(* IEC 61131-3 sources: plc_simulator/services/codesys/POUs, 112 files *)

(* ---- DEP_CalcIdleSlots.st ---- *)
(* ===========================================================================================
 *  DEP_CalcIdleSlots — Idle slot calculation per transporter
 *
 *  Company : Galvatek part of the John Cockerill Group
 *  Author  : Jarmo Piipponen
 *  Created : 25.03.2026
 *
 * -------------------------------------------------------------------------------------------
 *  Reads task queue via VAR_IN_OUT (sandbox or live).
 *  Writes idle slot sets to io_idle_slot per transporter.
 *
 *  ------------------------------------------------------------------------------------------
 *
 *  Changes:
 *
 *
 *
 *)

FUNCTION DEP_CalcIdleSlots : BOOL

(* Introduction of Variables ----------------------------------------------------------------*)

VAR_INPUT
  i_trans                   : INT;
  i_time_s                  : LINT;
END_VAR

VAR_IN_OUT  (* array sizes must match GVL_JC_Constants: 3=MAX_TRANSPORTERS *)
  io_task                   : ARRAY[1..3] OF UDT_JC_TskQueueType;
  io_idle_slot              : ARRAY[1..3] OF UDT_JC_DepIdleSlotSetType;
END_VAR

VAR_EXTERNAL CONSTANT
    MAX_TRANSPORTERS        : INT;
    MAX_UNITS               : INT;
    DEP_MAX_IDLE_SLOTS      : INT;
END_VAR

VAR_EXTERNAL
  g_transporter             : ARRAY[1..MAX_TRANSPORTERS] OF UDT_TransporterStatusType;
END_VAR

VAR
  qi                        : INT;
  si                        : INT;
  cnt                       : INT;
  prev_end                  : LINT;
  prev_sink                 : INT;
  gap_start                 : LINT;
  gap_end                   : LINT;
  HORIZON                   : LINT := 9999999999;
END_VAR

DEP_CalcIdleSlots := FALSE;
IF i_trans < 1 OR i_trans > MAX_TRANSPORTERS THEN RETURN; END_IF;

io_idle_slot[i_trans].Count := 0;
si := 0;
cnt := io_task[i_trans].Count;

prev_end  := i_time_s;
prev_sink := g_transporter[i_trans].CurrentStation;

FOR qi := 1 TO MAX_UNITS DO
  IF qi > cnt THEN EXIT; END_IF;

  gap_start := prev_end;
  gap_end   := io_task[i_trans].Queue[qi].StartTime;

  IF gap_end > gap_start + LINT#1 THEN
    si := si + 1;
    IF si <= DEP_MAX_IDLE_SLOTS THEN
      io_idle_slot[i_trans].Slots[si].StartTime   := gap_start;
      io_idle_slot[i_trans].Slots[si].EndTime     := gap_end;
      io_idle_slot[i_trans].Slots[si].LiftStationTarget := prev_sink;
      io_idle_slot[i_trans].Slots[si].SinkStationTarget := io_task[i_trans].Queue[qi].LiftStationTarget;
    END_IF;
  END_IF;

  prev_end  := io_task[i_trans].Queue[qi].FinishTime;
  prev_sink := io_task[i_trans].Queue[qi].SinkStationTarget;
END_FOR;

si := si + 1;
IF si <= DEP_MAX_IDLE_SLOTS THEN
  io_idle_slot[i_trans].Slots[si].StartTime   := prev_end;
  io_idle_slot[i_trans].Slots[si].EndTime     := HORIZON;
  io_idle_slot[i_trans].Slots[si].LiftStationTarget := prev_sink;
  io_idle_slot[i_trans].Slots[si].SinkStationTarget := 0;
END_IF;

io_idle_slot[i_trans].Count := si;
DEP_CalcIdleSlots := TRUE;

END_FUNCTION

(* ---- DEP_CalcOverlap.st ---- *)
(* ===========================================================================================
 *  DEP_CalcOverlap — Overlap station detection
 *
 *  Company : Galvatek part of the John Cockerill Group
 *  Author  : Jarmo Piipponen
 *  Created : 25.03.2026
 *
 * -------------------------------------------------------------------------------------------
 *  Identifies stations covered by 2+ transporters.
 *  Reads Transporters (read-only config). Writes io_overlap.
 *
 *  ------------------------------------------------------------------------------------------
 *
 *  Changes:
 *
 *
 *
 *)

FUNCTION DEP_CalcOverlap : BOOL

(* Introduction of Variables ----------------------------------------------------------------*)

VAR_IN_OUT
  io_overlap                : UDT_JC_DepOverlapType;
END_VAR

VAR_EXTERNAL CONSTANT
    MAX_TRANSPORTERS        : INT;
    MIN_STATION_INDEX        : INT;
    MAX_STATION_INDEX        : INT;
END_VAR

VAR_EXTERNAL
  Transporters                     : ARRAY[0..MAX_TRANSPORTERS] OF UDT_TransporterType;
END_VAR

VAR
  station_idx               : INT;
  ti                        : INT;
  ai                        : INT;
  cover_count               : INT;
  covered                   : BOOL;
  area                      : UDT_TaskArea;
END_VAR

io_overlap.Count := 0;

FOR station_idx := 0 TO 200 DO
  io_overlap.Flags[station_idx] := FALSE;
END_FOR;

FOR station_idx := MIN_STATION_INDEX TO MAX_STATION_INDEX DO
  cover_count := 0;

  FOR ti := 1 TO MAX_TRANSPORTERS DO
    covered := FALSE;
    FOR ai := 1 TO 4 DO
      IF NOT covered THEN
        area := Transporters[ti].TaskArea[ai];
        IF (area.MinLift > 0 AND station_idx >= area.MinLift AND station_idx <= area.MaxLift)
           OR (area.MinSink > 0 AND station_idx >= area.MinSink AND station_idx <= area.MaxSink) THEN
          covered := TRUE;
        END_IF;
      END_IF;
    END_FOR;
    IF covered THEN
      cover_count := cover_count + 1;
    END_IF;
  END_FOR;

  IF cover_count >= 2 THEN
    io_overlap.Flags[station_idx] := TRUE;
    io_overlap.Count := io_overlap.Count + 1;
  END_IF;
END_FOR;

DEP_CalcOverlap := TRUE;

END_FUNCTION

(* ---- DEP_FC_CalcIdleSlots.st ---- *)
(* ===========================================================================================
 *  DEP_FC_CalcIdleSlots — Idle slot calculation per transporter
 *
 *  Company : Galvatek part of the John Cockerill Group
 *  Author  : Jarmo Piipponen
 *  Created : 25.03.2026
 *
 * -------------------------------------------------------------------------------------------
 *  Reads task queue via VAR_IN_OUT (sandbox or live).
 *  Writes idle slot sets to ioIdleSlot per transporter.
 *
 *  ------------------------------------------------------------------------------------------
 *
 *  Changes:
 *
 *
 *
 *)

FUNCTION DEP_FC_CalcIdleSlots : BOOL

(* Introduction of Variables ----------------------------------------------------------------*)

VAR_INPUT
  iTrans                   : INT;
  iTimeS                  : LINT;
END_VAR

VAR_IN_OUT  (* array sizes must match GVL_JC_Constants: 3=MAX_TRANSPORTERS *)
  ioTask                   : ARRAY[1..3] OF UDT_JC_TskQueueType;
  ioIdleSlot              : ARRAY[1..3] OF UDT_JC_DepIdleSlotSetType;
END_VAR

VAR_EXTERNAL CONSTANT
    MAX_TRANSPORTERS        : INT;
    MAX_UNITS               : INT;
    DEP_MAX_IDLE_SLOTS      : INT;
END_VAR

VAR_EXTERNAL
  TransporterStatus             : ARRAY[1..MAX_TRANSPORTERS] OF UDT_TransporterStatusType;
END_VAR

VAR
  vQi                        : INT;
  vSi                        : INT;
  vCnt                       : INT;
  vPrevEnd                  : LINT;
  vPrevSink                 : INT;
  vGapStart                 : LINT;
  vGapEnd                   : LINT;
  vHorizon                   : LINT := 9999999999;
END_VAR

DEP_FC_CalcIdleSlots := FALSE;
IF iTrans < 1 OR iTrans > MAX_TRANSPORTERS THEN RETURN; END_IF;

ioIdleSlot[iTrans].Count := 0;
vSi := 0;
vCnt := ioTask[iTrans].Count;

vPrevEnd  := iTimeS;
vPrevSink := TransporterStatus[iTrans].CurrentStation;

FOR vQi := 1 TO MAX_UNITS DO
  IF vQi > vCnt THEN EXIT; END_IF;

  vGapStart := vPrevEnd;
  vGapEnd   := ioTask[iTrans].Queue[vQi].StartTime;

  IF vGapEnd > vGapStart + LINT#1 THEN
    vSi := vSi + 1;
    IF vSi <= DEP_MAX_IDLE_SLOTS THEN
      ioIdleSlot[iTrans].Slots[vSi].StartTime   := vGapStart;
      ioIdleSlot[iTrans].Slots[vSi].EndTime     := vGapEnd;
      ioIdleSlot[iTrans].Slots[vSi].LiftStationTarget := vPrevSink;
      ioIdleSlot[iTrans].Slots[vSi].SinkStationTarget := ioTask[iTrans].Queue[vQi].LiftStationTarget;
    END_IF;
  END_IF;

  vPrevEnd  := ioTask[iTrans].Queue[vQi].FinishTime;
  vPrevSink := ioTask[iTrans].Queue[vQi].SinkStationTarget;
END_FOR;

vSi := vSi + 1;
IF vSi <= DEP_MAX_IDLE_SLOTS THEN
  ioIdleSlot[iTrans].Slots[vSi].StartTime   := vPrevEnd;
  ioIdleSlot[iTrans].Slots[vSi].EndTime     := vHorizon;
  ioIdleSlot[iTrans].Slots[vSi].LiftStationTarget := vPrevSink;
  ioIdleSlot[iTrans].Slots[vSi].SinkStationTarget := 0;
END_IF;

ioIdleSlot[iTrans].Count := vSi;
DEP_FC_CalcIdleSlots := TRUE;

END_FUNCTION

(* ---- DEP_FC_CalcOverlap.st ---- *)
(* ===========================================================================================
 *  DEP_FC_CalcOverlap — Overlap station detection
 *
 *  Company : Galvatek part of the John Cockerill Group
 *  Author  : Jarmo Piipponen
 *  Created : 25.03.2026
 *
 * -------------------------------------------------------------------------------------------
 *  Identifies stations vCovered by 2+ transporters.
 *  Reads Transporters (read-only config). Writes ioOverlap.
 *
 *  ------------------------------------------------------------------------------------------
 *
 *  Changes:
 *
 *
 *
 *)

FUNCTION DEP_FC_CalcOverlap : BOOL

(* Introduction of Variables ----------------------------------------------------------------*)

VAR_IN_OUT
  ioOverlap                : UDT_JC_DepOverlapType;
END_VAR

VAR_EXTERNAL CONSTANT
    MAX_TRANSPORTERS        : INT;
    MIN_STATION_INDEX        : INT;
    MAX_STATION_INDEX        : INT;
END_VAR

VAR_EXTERNAL
  Transporters                     : ARRAY[0..MAX_TRANSPORTERS] OF UDT_TransporterType;
END_VAR

VAR
  vStationIdx               : INT;
  vTi                        : INT;
  vAi                        : INT;
  vCoverCount               : INT;
  vCovered                   : BOOL;
  vArea                      : UDT_TaskAreaType;
END_VAR

ioOverlap.Count := 0;

FOR vStationIdx := 0 TO 200 DO
  ioOverlap.Flags[vStationIdx] := FALSE;
END_FOR;

FOR vStationIdx := MIN_STATION_INDEX TO MAX_STATION_INDEX DO
  vCoverCount := 0;

  FOR vTi := 1 TO MAX_TRANSPORTERS DO
    vCovered := FALSE;
    FOR vAi := 1 TO 4 DO
      IF NOT vCovered THEN
        vArea := Transporters[vTi].TaskArea[vAi];
        IF (vArea.MinLift > 0 AND vStationIdx >= vArea.MinLift AND vStationIdx <= vArea.MaxLift)
           OR (vArea.MinSink > 0 AND vStationIdx >= vArea.MinSink AND vStationIdx <= vArea.MaxSink) THEN
          vCovered := TRUE;
        END_IF;
      END_IF;
    END_FOR;
    IF vCovered THEN
      vCoverCount := vCoverCount + 1;
    END_IF;
  END_FOR;

  IF vCoverCount >= 2 THEN
    ioOverlap.Flags[vStationIdx] := TRUE;
    ioOverlap.Count := ioOverlap.Count + 1;
  END_IF;
END_FOR;

DEP_FC_CalcOverlap := TRUE;

END_FUNCTION

(* ---- DEP_FC_FitTaskToSlot.st ---- *)
(* ===========================================================================================
 *  DEP_FC_FitTaskToSlot — Fit a departure task into idle slots
 *
 *  Company : Galvatek part of the John Cockerill Group
 *  Author  : Jarmo Piipponen
 *  Created : 25.03.2026
 *
 * -------------------------------------------------------------------------------------------
 *  Reads idle slots and move times.
 *  Returns fit result via VAR_OUTPUT.
 *
 *  ------------------------------------------------------------------------------------------
 *
 *  Changes:
 *
 *
 *
 *)

FUNCTION DEP_FC_FitTaskToSlot : BOOL

(* Introduction of Variables ----------------------------------------------------------------*)

VAR_INPUT
  iLiftStn                : INT;
  iSinkStn                : INT;
  iTransId                : INT;
  iTaskStart              : LINT;
  iTaskEnd                : LINT;
  iShiftS                 : REAL;
  iCalcTimeS             : DINT;
  iMinTimeS              : DINT;
  iMaxTimeS              : DINT;
  iFlexFactor             : REAL;
  iMarginS                : REAL;
  iConflictMarginS       : REAL;
END_VAR

VAR_IN_OUT  (* array sizes must match GVL_JC_Constants: 3=MAX_TRANSPORTERS *)
  ioIdleSlot              : ARRAY[1..3] OF UDT_JC_DepIdleSlotSetType;
  ioOResult                  : UDT_JC_DepFitResultType;
END_VAR

VAR_EXTERNAL CONSTANT
    MAX_TRANSPORTERS        : INT;
    DEP_MAX_IDLE_SLOTS      : INT;
    SCH_DISPATCH_MARGIN_S   : REAL;
END_VAR

VAR_EXTERNAL
  Move                    : ARRAY[1..MAX_TRANSPORTERS] OF UDT_JC_MoveTimesType;
END_VAR

VAR
  vSi                        : INT;
  vSlotCnt                  : INT;
  vSlotStart                : LINT;
  vSlotEnd                  : LINT;
  vFromStn                  : INT;
  vToStn                    : INT;
  vTravelTo                 : REAL;
  vTravelFrom               : REAL;
  vEarliest                  : LINT;
  vLatest                    : LINT;
  vTaskDur                  : LINT;
  vDelay                     : REAL;
  vFlexUp                   : REAL;
  vCappedFlex               : REAL;
  vBestDelay                : REAL;
  vBestSlot                 : INT;
  vFound                     : BOOL;
  vOverflowBestDelay       : REAL;
  vOverflowBestSlot        : INT;
  vTmpMove                  : UDT_JC_MoveTimesType;
  vTotalDelay               : REAL;
END_VAR

ioOResult.Fits         := FALSE;
ioOResult.DelayTime    := 0;
ioOResult.NeedExtraTime := 0;
ioOResult.TaskEndTime  := 0;
ioOResult.SlotIdx      := 0;
ioOResult.OverflowSlotIdx := 0;
ioOResult.TransporterId := iTransId;
DEP_FC_FitTaskToSlot := FALSE;

IF iTransId < 1 OR iTransId > MAX_TRANSPORTERS THEN RETURN; END_IF;

vTaskDur   := iTaskEnd - iTaskStart;
(* Absolute cap: flex based on full (max - min) range, not (max - calc).
   This prevents cumulative drift when CalcTime is adjusted across rounds. *)
vFlexUp    := DINT_TO_REAL(iMaxTimeS - iMinTimeS);
  IF vFlexUp < 0.0 THEN vFlexUp := 0.0; END_IF;
vCappedFlex := vFlexUp * iFlexFactor;

vSlotCnt   := ioIdleSlot[iTransId].Count;
vBestDelay := 1.0E9;
vBestSlot  := 0;
vFound      := FALSE;
vOverflowBestDelay := 1.0E9;
vOverflowBestSlot  := 0;

vTmpMove := Move[iTransId];
FOR vSi := 1 TO DEP_MAX_IDLE_SLOTS DO
  IF vSi > vSlotCnt THEN EXIT; END_IF;

  vSlotStart := ioIdleSlot[iTransId].Slots[vSi].StartTime;
  vSlotEnd   := ioIdleSlot[iTransId].Slots[vSi].EndTime;

  vFromStn := ioIdleSlot[iTransId].Slots[vSi].LiftStationTarget;
  vTravelTo := 0.0;
  IF vFromStn > 0 AND vFromStn <> iLiftStn THEN
    vTravelTo := STC_FC_CalcHorizontalTravel(iFromStn := vFromStn, iToStn := iLiftStn, iMove := vTmpMove);
  END_IF;

  vToStn := ioIdleSlot[iTransId].Slots[vSi].SinkStationTarget;
  vTravelFrom := 0.0;
  IF vToStn > 0 AND vToStn <> iSinkStn THEN
    vTravelFrom := STC_FC_CalcHorizontalTravel(iFromStn := iSinkStn, iToStn := vToStn, iMove := vTmpMove);
  END_IF;

  (* vEarliest = max(transporter arrival, task readiness) + conflict margin *)
  IF (vSlotStart + REAL_TO_LINT(vTravelTo)) > (iTaskStart + REAL_TO_LINT(iShiftS)) THEN
    vEarliest := vSlotStart + REAL_TO_LINT(vTravelTo + iConflictMarginS);
  ELSE
    vEarliest := iTaskStart + REAL_TO_LINT(iShiftS + iConflictMarginS);
  END_IF;

  IF vSlotEnd > LINT#9000000000 THEN
    vLatest := LINT#9000000000;
  ELSE
    vLatest := vSlotEnd - REAL_TO_LINT(vTravelFrom + SCH_DISPATCH_MARGIN_S);
  END_IF;

  IF vEarliest + vTaskDur <= vLatest THEN
    vDelay := LINT_TO_REAL(vEarliest - iTaskStart) - iShiftS;
  IF vDelay < 0.0 THEN vDelay := 0.0; END_IF;
    vTotalDelay := iShiftS + vDelay;

    IF vTotalDelay <= iMarginS OR vTotalDelay <= vCappedFlex + 1.0 THEN
      IF vDelay < vBestDelay THEN
        vBestDelay := vDelay;
        vBestSlot  := vSi;
        vFound      := TRUE;
      END_IF;
    ELSE
      IF vDelay < vOverflowBestDelay THEN
        vOverflowBestDelay := vDelay;
        vOverflowBestSlot  := vSi;
      END_IF;
    END_IF;
  END_IF;
END_FOR;

IF vFound THEN
  ioOResult.Fits      := TRUE;
  ioOResult.DelayTime := REAL_TO_DINT(vBestDelay);
  ioOResult.SlotIdx   := vBestSlot;
  ioOResult.TaskEndTime := iTaskStart + REAL_TO_LINT(iShiftS + vBestDelay) + vTaskDur;
  ioOResult.NeedExtraTime := 0;
ELSE
  ioOResult.Fits := FALSE;
  IF vOverflowBestDelay < 1.0E8 THEN
    ioOResult.DelayTime     := REAL_TO_DINT(vOverflowBestDelay);
    ioOResult.NeedExtraTime := REAL_TO_DINT(iShiftS + vOverflowBestDelay - vCappedFlex);
  IF ioOResult.NeedExtraTime < 0 THEN ioOResult.NeedExtraTime := 0; END_IF;
    ioOResult.OverflowSlotIdx := vOverflowBestSlot;
  ELSE
    ioOResult.NeedExtraTime := 0;
  END_IF;
END_IF;

DEP_FC_FitTaskToSlot := TRUE;

END_FUNCTION

(* ---- DEP_FC_OverlapDelay.st ---- *)
(* ===========================================================================================
 *  DEP_FC_OverlapDelay — Overlap conflict vDelay calculation
 *
 *  Company : Galvatek part of the John Cockerill Group
 *  Author  : Jarmo Piipponen
 *  Created : 25.03.2026
 *
 * -------------------------------------------------------------------------------------------
 *  Returns vDelay vNeeded to avoid overlap conflicts.
 *  Reads task queues via ioTask (sandbox or live).
 *
 *  ------------------------------------------------------------------------------------------
 *
 *  Changes:
 *
 *
 *
 *)

FUNCTION DEP_FC_OverlapDelay : REAL   (* returns delay_s, 0 = no conflict *)

(* Introduction of Variables ----------------------------------------------------------------*)

VAR_INPUT
  iLiftStn                : INT;
  iSinkStn                : INT;
  iTransId                : INT;
  iTaskStart              : LINT;
  iTaskEnd                : LINT;
  iMarginS                : REAL;
END_VAR

VAR_IN_OUT  (* array sizes must match GVL_JC_Constants: 3=MAX_TRANSPORTERS *)
  ioTask                   : ARRAY[1..3] OF UDT_JC_TskQueueType;
  ioOverlap                : UDT_JC_DepOverlapType;
END_VAR

VAR_EXTERNAL CONSTANT
    MAX_TRANSPORTERS        : INT;
    MAX_UNITS               : INT;
    DEP_MAX_DELAY_ACTS      : INT;
END_VAR

VAR
  vLiftIsOverlap           : BOOL;
  vSinkIsOverlap           : BOOL;
  vRound                     : INT;
  vTi                        : INT;
  vQi                        : INT;
  vMaxConf                  : REAL;
  vTStart                   : LINT;
  vTEnd                     : LINT;
  vEStart                   : LINT;
  vEEnd                     : LINT;
  vELift                    : INT;
  vESink                    : INT;
  vHasOvlp                  : BOOL;
  vNeeded                    : REAL;
  vDelay                     : REAL;
END_VAR

vDelay := 0.0;

IF iLiftStn >= 0 AND iLiftStn <= 200 THEN
  vLiftIsOverlap := ioOverlap.Flags[iLiftStn];
ELSE
  vLiftIsOverlap := FALSE;
END_IF;
IF iSinkStn >= 0 AND iSinkStn <= 200 THEN
  vSinkIsOverlap := ioOverlap.Flags[iSinkStn];
ELSE
  vSinkIsOverlap := FALSE;
END_IF;

IF NOT vLiftIsOverlap AND NOT vSinkIsOverlap THEN
  DEP_FC_OverlapDelay := 0.0;
  RETURN;
END_IF;

FOR vRound := 1 TO DEP_MAX_DELAY_ACTS DO
  vMaxConf := 0.0;
  vTStart  := iTaskStart + REAL_TO_LINT(vDelay);
  vTEnd    := iTaskEnd + REAL_TO_LINT(vDelay);

  FOR vTi := 1 TO MAX_TRANSPORTERS DO
    IF vTi <> iTransId THEN
      FOR vQi := 1 TO MAX_UNITS DO
        IF vQi > ioTask[vTi].Count THEN EXIT; END_IF;

        vELift  := ioTask[vTi].Queue[vQi].LiftStationTarget;
        vESink  := ioTask[vTi].Queue[vQi].SinkStationTarget;
        vEStart := ioTask[vTi].Queue[vQi].StartTime;
        vEEnd   := ioTask[vTi].Queue[vQi].FinishTime;

        vHasOvlp := FALSE;
        IF vELift >= 0 AND vELift <= 200 THEN
  IF ioOverlap.Flags[vELift] THEN vHasOvlp := TRUE; END_IF;
        END_IF;
        IF NOT vHasOvlp AND vESink >= 0 AND vESink <= 200 THEN
  IF ioOverlap.Flags[vESink] THEN vHasOvlp := TRUE; END_IF;
        END_IF;

        IF vHasOvlp THEN
          IF vTStart < (vEEnd + REAL_TO_LINT(iMarginS)) AND vTEnd > (vEStart - REAL_TO_LINT(iMarginS)) THEN
            vNeeded := LINT_TO_REAL(vEEnd - vTStart) + iMarginS;
  IF vNeeded > vMaxConf THEN vMaxConf := vNeeded; END_IF;
          END_IF;
        END_IF;

      END_FOR;
    END_IF;
  END_FOR;

  IF vMaxConf <= 0.0 THEN EXIT; END_IF;
  vDelay := vDelay + vMaxConf;
END_FOR;

DEP_FC_OverlapDelay := vDelay;

END_FUNCTION

(* ---- DEP_FC_Sandbox.st ---- *)
(* ===========================================================================================
 *  DEP_FC_Sandbox — Sandbox snapshot / restore / clear
 *
 *  Company : Galvatek part of the John Cockerill Group
 *  Author  : Jarmo Piipponen
 *  Created : 25.03.2026
 *
 * -------------------------------------------------------------------------------------------
 *  Copies batch and program data between live globals and
 *  DEP workspace arrays via VAR_IN_OUT.
 *  Schedule is NOT copied — DEP calculates it fresh (phases 1000+i).
 *  Task queues are NOT copied — DEP rebuilds them (phases 2000+).
 *
 *  Commands:
 *  1 = SNAPSHOT  — live batch+program → workspace
 *  2 = RESTORE   — workspace batch+program → live
 *  3 = CLEAR     — noop for array-based workspace
 *
 *  ------------------------------------------------------------------------------------------
 *
 *  Changes:
 *
 *
 *
 *)

FUNCTION DEP_FC_Sandbox : BOOL

(* Introduction of Variables ----------------------------------------------------------------*)

VAR_INPUT
  iCmd                     : INT;
END_VAR

VAR_IN_OUT  (* array sizes must match GVL_JC_Constants: 10=MAX_UNITS, 3=MAX_TRANSPORTERS *)
  ioWkSchedule            : ARRAY[1..10] OF UDT_JC_TskScheduleType;
  ioWkBatch               : ARRAY[1..10] OF UDT_BatchType;
  ioWkProgram             : ARRAY[1..10] OF UDT_TreatmentProgramType;
  ioWkTask                : ARRAY[1..3] OF UDT_JC_TskQueueType;
END_VAR

VAR_EXTERNAL CONSTANT
    MAX_TRANSPORTERS        : INT;
    MAX_UNITS               : INT;
END_VAR

VAR_EXTERNAL
  Schedule                : ARRAY[1..MAX_UNITS] OF UDT_JC_TskScheduleType;
  Batch                   : ARRAY[1..MAX_UNITS] OF UDT_BatchType;
  TreatmentPrograms                 : ARRAY[1..MAX_UNITS] OF UDT_TreatmentProgramType;
  Task                    : ARRAY[1..MAX_TRANSPORTERS] OF UDT_JC_TskQueueType;
END_VAR

VAR
  vUi                        : INT;
END_VAR

DEP_FC_Sandbox := TRUE;

IF iCmd = 1 THEN
  (* SNAPSHOT: clear workspace, then copy live batch+program *)
  FOR vUi := 1 TO MAX_UNITS DO
    ioWkSchedule[vUi].StageCount := 0;
    ioWkBatch[vUi]    := Batch[vUi];
    ioWkProgram[vUi]  := TreatmentPrograms[vUi];
  END_FOR;
  FOR vUi := 1 TO MAX_TRANSPORTERS DO
    ioWkTask[vUi].Count := 0;
  END_FOR;
ELSIF iCmd = 2 THEN
  (* RESTORE: workspace batch+program → live (for REJECT rollback) *)
  FOR vUi := 1 TO MAX_UNITS DO
    IF ioWkBatch[vUi].BatchCode > 0 THEN
      Batch[vUi] := ioWkBatch[vUi];
    END_IF;
    IF ioWkProgram[vUi].ProgramId > 0 THEN
      TreatmentPrograms[vUi] := ioWkProgram[vUi];
    END_IF;
  END_FOR;
ELSIF iCmd = 3 THEN
  ;  (* CLEAR: nothing needed *)

END_IF;

END_FUNCTION

(* ---- DEP_FitTaskToSlot.st ---- *)
(* ===========================================================================================
 *  DEP_FitTaskToSlot — Fit a departure task into idle slots
 *
 *  Company : Galvatek part of the John Cockerill Group
 *  Author  : Jarmo Piipponen
 *  Created : 25.03.2026
 *
 * -------------------------------------------------------------------------------------------
 *  Reads idle slots and move times.
 *  Returns fit result via VAR_OUTPUT.
 *
 *  ------------------------------------------------------------------------------------------
 *
 *  Changes:
 *
 *
 *
 *)

FUNCTION DEP_FitTaskToSlot : BOOL

(* Introduction of Variables ----------------------------------------------------------------*)

VAR_INPUT
  i_lift_stn                : INT;
  i_sink_stn                : INT;
  i_trans_id                : INT;
  i_task_start              : LINT;
  i_task_end                : LINT;
  i_shift_s                 : REAL;
  i_calc_time_s             : DINT;
  i_min_time_s              : DINT;
  i_max_time_s              : DINT;
  i_flex_factor             : REAL;
  i_margin_s                : REAL;
  i_conflict_margin_s       : REAL;
END_VAR

VAR_IN_OUT  (* array sizes must match GVL_JC_Constants: 3=MAX_TRANSPORTERS *)
  io_idle_slot              : ARRAY[1..3] OF UDT_JC_DepIdleSlotSetType;
  o_result                  : UDT_JC_DepFitResultType;
END_VAR

VAR_EXTERNAL CONSTANT
    MAX_TRANSPORTERS        : INT;
    DEP_MAX_IDLE_SLOTS      : INT;
    SCH_DISPATCH_MARGIN_S   : REAL;
END_VAR

VAR_EXTERNAL
  g_move                    : ARRAY[1..MAX_TRANSPORTERS] OF UDT_JC_MoveTimesType;
END_VAR

VAR
  si                        : INT;
  slot_cnt                  : INT;
  slot_start                : LINT;
  slot_end                  : LINT;
  from_stn                  : INT;
  to_stn                    : INT;
  travel_to                 : REAL;
  travel_from               : REAL;
  earliest                  : LINT;
  latest                    : LINT;
  task_dur                  : LINT;
  delay                     : REAL;
  flex_up                   : REAL;
  capped_flex               : REAL;
  best_delay                : REAL;
  best_slot                 : INT;
  found                     : BOOL;
  overflow_best_delay       : REAL;
  overflow_best_slot        : INT;
  tmp_move                  : UDT_JC_MoveTimesType;
  total_delay               : REAL;
END_VAR

o_result.Fits         := FALSE;
o_result.DelayTime    := 0;
o_result.NeedExtraTime := 0;
o_result.TaskEndTime  := 0;
o_result.SlotIdx      := 0;
o_result.OverflowSlotIdx := 0;
o_result.TransporterId := i_trans_id;
DEP_FitTaskToSlot := FALSE;

IF i_trans_id < 1 OR i_trans_id > MAX_TRANSPORTERS THEN RETURN; END_IF;

task_dur   := i_task_end - i_task_start;
(* Absolute cap: flex based on full (max - min) range, not (max - calc).
   This prevents cumulative drift when CalcTime is adjusted across rounds. *)
flex_up    := DINT_TO_REAL(i_max_time_s - i_min_time_s);
  IF flex_up < 0.0 THEN flex_up := 0.0; END_IF;
capped_flex := flex_up * i_flex_factor;

slot_cnt   := io_idle_slot[i_trans_id].Count;
best_delay := 1.0E9;
best_slot  := 0;
found      := FALSE;
overflow_best_delay := 1.0E9;
overflow_best_slot  := 0;

tmp_move := g_move[i_trans_id];
FOR si := 1 TO DEP_MAX_IDLE_SLOTS DO
  IF si > slot_cnt THEN EXIT; END_IF;

  slot_start := io_idle_slot[i_trans_id].Slots[si].StartTime;
  slot_end   := io_idle_slot[i_trans_id].Slots[si].EndTime;

  from_stn := io_idle_slot[i_trans_id].Slots[si].LiftStationTarget;
  travel_to := 0.0;
  IF from_stn > 0 AND from_stn <> i_lift_stn THEN
    travel_to := STC_CalcHorizontalTravel(i_from_stn := from_stn, i_to_stn := i_lift_stn, i_move := tmp_move);
  END_IF;

  to_stn := io_idle_slot[i_trans_id].Slots[si].SinkStationTarget;
  travel_from := 0.0;
  IF to_stn > 0 AND to_stn <> i_sink_stn THEN
    travel_from := STC_CalcHorizontalTravel(i_from_stn := i_sink_stn, i_to_stn := to_stn, i_move := tmp_move);
  END_IF;

  (* earliest = max(transporter arrival, task readiness) + conflict margin *)
  IF (slot_start + REAL_TO_LINT(travel_to)) > (i_task_start + REAL_TO_LINT(i_shift_s)) THEN
    earliest := slot_start + REAL_TO_LINT(travel_to + i_conflict_margin_s);
  ELSE
    earliest := i_task_start + REAL_TO_LINT(i_shift_s + i_conflict_margin_s);
  END_IF;

  IF slot_end > LINT#9000000000 THEN
    latest := LINT#9000000000;
  ELSE
    latest := slot_end - REAL_TO_LINT(travel_from + SCH_DISPATCH_MARGIN_S);
  END_IF;

  IF earliest + task_dur <= latest THEN
    delay := LINT_TO_REAL(earliest - i_task_start) - i_shift_s;
  IF delay < 0.0 THEN delay := 0.0; END_IF;
    total_delay := i_shift_s + delay;

    IF total_delay <= i_margin_s OR total_delay <= capped_flex + 1.0 THEN
      IF delay < best_delay THEN
        best_delay := delay;
        best_slot  := si;
        found      := TRUE;
      END_IF;
    ELSE
      IF delay < overflow_best_delay THEN
        overflow_best_delay := delay;
        overflow_best_slot  := si;
      END_IF;
    END_IF;
  END_IF;
END_FOR;

IF found THEN
  o_result.Fits      := TRUE;
  o_result.DelayTime := REAL_TO_DINT(best_delay);
  o_result.SlotIdx   := best_slot;
  o_result.TaskEndTime := i_task_start + REAL_TO_LINT(i_shift_s + best_delay) + task_dur;
  o_result.NeedExtraTime := 0;
ELSE
  o_result.Fits := FALSE;
  IF overflow_best_delay < 1.0E8 THEN
    o_result.DelayTime     := REAL_TO_DINT(overflow_best_delay);
    o_result.NeedExtraTime := REAL_TO_DINT(i_shift_s + overflow_best_delay - capped_flex);
  IF o_result.NeedExtraTime < 0 THEN o_result.NeedExtraTime := 0; END_IF;
    o_result.OverflowSlotIdx := overflow_best_slot;
  ELSE
    o_result.NeedExtraTime := 0;
  END_IF;
END_IF;

DEP_FitTaskToSlot := TRUE;

END_FUNCTION

(* ---- DEP_OverlapDelay.st ---- *)
(* ===========================================================================================
 *  DEP_OverlapDelay — Overlap conflict delay calculation
 *
 *  Company : Galvatek part of the John Cockerill Group
 *  Author  : Jarmo Piipponen
 *  Created : 25.03.2026
 *
 * -------------------------------------------------------------------------------------------
 *  Returns delay needed to avoid overlap conflicts.
 *  Reads task queues via io_task (sandbox or live).
 *
 *  ------------------------------------------------------------------------------------------
 *
 *  Changes:
 *
 *
 *
 *)

FUNCTION DEP_OverlapDelay : REAL   (* returns delay_s, 0 = no conflict *)

(* Introduction of Variables ----------------------------------------------------------------*)

VAR_INPUT
  i_lift_stn                : INT;
  i_sink_stn                : INT;
  i_trans_id                : INT;
  i_task_start              : LINT;
  i_task_end                : LINT;
  i_margin_s                : REAL;
END_VAR

VAR_IN_OUT  (* array sizes must match GVL_JC_Constants: 3=MAX_TRANSPORTERS *)
  io_task                   : ARRAY[1..3] OF UDT_JC_TskQueueType;
  io_overlap                : UDT_JC_DepOverlapType;
END_VAR

VAR_EXTERNAL CONSTANT
    MAX_TRANSPORTERS        : INT;
    MAX_UNITS               : INT;
    DEP_MAX_DELAY_ACTS      : INT;
END_VAR

VAR
  lift_is_overlap           : BOOL;
  sink_is_overlap           : BOOL;
  round                     : INT;
  ti                        : INT;
  qi                        : INT;
  max_conf                  : REAL;
  t_start                   : LINT;
  t_end                     : LINT;
  e_start                   : LINT;
  e_end                     : LINT;
  e_lift                    : INT;
  e_sink                    : INT;
  has_ovlp                  : BOOL;
  needed                    : REAL;
  delay                     : REAL;
END_VAR

delay := 0.0;

IF i_lift_stn >= 0 AND i_lift_stn <= 200 THEN
  lift_is_overlap := io_overlap.Flags[i_lift_stn];
ELSE
  lift_is_overlap := FALSE;
END_IF;
IF i_sink_stn >= 0 AND i_sink_stn <= 200 THEN
  sink_is_overlap := io_overlap.Flags[i_sink_stn];
ELSE
  sink_is_overlap := FALSE;
END_IF;

IF NOT lift_is_overlap AND NOT sink_is_overlap THEN
  DEP_OverlapDelay := 0.0;
  RETURN;
END_IF;

FOR round := 1 TO DEP_MAX_DELAY_ACTS DO
  max_conf := 0.0;
  t_start  := i_task_start + REAL_TO_LINT(delay);
  t_end    := i_task_end + REAL_TO_LINT(delay);

  FOR ti := 1 TO MAX_TRANSPORTERS DO
    IF ti <> i_trans_id THEN
      FOR qi := 1 TO MAX_UNITS DO
        IF qi > io_task[ti].Count THEN EXIT; END_IF;

        e_lift  := io_task[ti].Queue[qi].LiftStationTarget;
        e_sink  := io_task[ti].Queue[qi].SinkStationTarget;
        e_start := io_task[ti].Queue[qi].StartTime;
        e_end   := io_task[ti].Queue[qi].FinishTime;

        has_ovlp := FALSE;
        IF e_lift >= 0 AND e_lift <= 200 THEN
  IF io_overlap.Flags[e_lift] THEN has_ovlp := TRUE; END_IF;
        END_IF;
        IF NOT has_ovlp AND e_sink >= 0 AND e_sink <= 200 THEN
  IF io_overlap.Flags[e_sink] THEN has_ovlp := TRUE; END_IF;
        END_IF;

        IF has_ovlp THEN
          IF t_start < (e_end + REAL_TO_LINT(i_margin_s)) AND t_end > (e_start - REAL_TO_LINT(i_margin_s)) THEN
            needed := LINT_TO_REAL(e_end - t_start) + i_margin_s;
  IF needed > max_conf THEN max_conf := needed; END_IF;
          END_IF;
        END_IF;

      END_FOR;
    END_IF;
  END_FOR;

  IF max_conf <= 0.0 THEN EXIT; END_IF;
  delay := delay + max_conf;
END_FOR;

DEP_OverlapDelay := delay;

END_FUNCTION

(* ---- DEP_Sandbox.st ---- *)
(* ===========================================================================================
 *  DEP_Sandbox — Sandbox snapshot / restore / clear
 *
 *  Company : Galvatek part of the John Cockerill Group
 *  Author  : Jarmo Piipponen
 *  Created : 25.03.2026
 *
 * -------------------------------------------------------------------------------------------
 *  Copies batch and program data between live globals and
 *  DEP workspace arrays via VAR_IN_OUT.
 *  Schedule is NOT copied — DEP calculates it fresh (phases 1000+i).
 *  Task queues are NOT copied — DEP rebuilds them (phases 2000+).
 *
 *  Commands:
 *  1 = SNAPSHOT  — live batch+program → workspace
 *  2 = RESTORE   — workspace batch+program → live
 *  3 = CLEAR     — noop for array-based workspace
 *
 *  ------------------------------------------------------------------------------------------
 *
 *  Changes:
 *
 *
 *
 *)

FUNCTION DEP_Sandbox : BOOL

(* Introduction of Variables ----------------------------------------------------------------*)

VAR_INPUT
  i_cmd                     : INT;
END_VAR

VAR_IN_OUT  (* array sizes must match GVL_JC_Constants: 10=MAX_UNITS, 3=MAX_TRANSPORTERS *)
  io_wk_schedule            : ARRAY[1..10] OF UDT_JC_TskScheduleType;
  io_wk_batch               : ARRAY[1..10] OF UDT_BatchType;
  io_wk_program             : ARRAY[1..10] OF UDT_TreatmentProgramType;
  io_wk_task                : ARRAY[1..3] OF UDT_JC_TskQueueType;
END_VAR

VAR_EXTERNAL CONSTANT
    MAX_TRANSPORTERS        : INT;
    MAX_UNITS               : INT;
END_VAR

VAR_EXTERNAL
  g_schedule                : ARRAY[1..MAX_UNITS] OF UDT_JC_TskScheduleType;
  g_batch                   : ARRAY[1..MAX_UNITS] OF UDT_BatchType;
  TreatmentPrograms                 : ARRAY[1..MAX_UNITS] OF UDT_TreatmentProgramType;
  g_task                    : ARRAY[1..MAX_TRANSPORTERS] OF UDT_JC_TskQueueType;
END_VAR

VAR
  ui                        : INT;
END_VAR

DEP_Sandbox := TRUE;

IF i_cmd = 1 THEN
  (* SNAPSHOT: clear workspace, then copy live batch+program *)
  FOR ui := 1 TO MAX_UNITS DO
    io_wk_schedule[ui].StageCount := 0;
    io_wk_batch[ui]    := g_batch[ui];
    io_wk_program[ui]  := TreatmentPrograms[ui];
  END_FOR;
  FOR ui := 1 TO MAX_TRANSPORTERS DO
    io_wk_task[ui].Count := 0;
  END_FOR;
ELSIF i_cmd = 2 THEN
  (* RESTORE: workspace batch+program → live (for REJECT rollback) *)
  FOR ui := 1 TO MAX_UNITS DO
    IF io_wk_batch[ui].BatchCode > 0 THEN
      g_batch[ui] := io_wk_batch[ui];
    END_IF;
    IF io_wk_program[ui].ProgramId > 0 THEN
      TreatmentPrograms[ui] := io_wk_program[ui];
    END_IF;
  END_FOR;
ELSIF i_cmd = 3 THEN
  ;  (* CLEAR: nothing needed *)

END_IF;

END_FUNCTION

(* ---- FC_DEP_CalcIdleSlots.st ---- *)
(* ===========================================================================================
 *  FC_DEP_CalcIdleSlots — Idle slot calculation per transporter
 *
 *  Company : Galvatek part of the John Cockerill Group
 *  Author  : Jarmo Piipponen
 *  Created : 25.03.2026
 *
 * -------------------------------------------------------------------------------------------
 *  Reads task queue via VAR_IN_OUT (sandbox or live).
 *  Writes idle slot sets to ioIdleSlot per transporter.
 *
 *  ------------------------------------------------------------------------------------------
 *
 *  Changes:
 *
 *
 *
 *)

FUNCTION FC_DEP_CalcIdleSlots : BOOL

(* Introduction of Variables ----------------------------------------------------------------*)

VAR_INPUT
  iTrans                   : INT;
  iTimeS                  : LINT;
END_VAR

VAR_IN_OUT  (* array sizes must match GVL_JC_Constants: 3=MAX_TRANSPORTERS *)
  ioTask                   : ARRAY[1..3] OF UDT_JC_TskQueueType;
  ioIdleSlot              : ARRAY[1..3] OF UDT_JC_DepIdleSlotSetType;
END_VAR

VAR_EXTERNAL CONSTANT
    MAX_TRANSPORTERS        : INT;
    MAX_UNITS               : INT;
    DEP_MAX_IDLE_SLOTS      : INT;
END_VAR

VAR_EXTERNAL
  g_transporter             : ARRAY[1..MAX_TRANSPORTERS] OF UDT_TransporterStatusType;
END_VAR

VAR
  qi                        : INT;
  si                        : INT;
  vCnt                       : INT;
  vPrevEnd                  : LINT;
  vPrevSink                 : INT;
  vGapStart                 : LINT;
  vGapEnd                   : LINT;
  HORIZON                   : LINT := 9999999999;
END_VAR

FC_DEP_CalcIdleSlots := FALSE;
IF iTrans < 1 OR iTrans > MAX_TRANSPORTERS THEN RETURN; END_IF;

ioIdleSlot[iTrans].Count := 0;
si := 0;
vCnt := ioTask[iTrans].Count;

vPrevEnd  := iTimeS;
vPrevSink := g_transporter[iTrans].CurrentStation;

FOR qi := 1 TO MAX_UNITS DO
  IF qi > vCnt THEN EXIT; END_IF;

  vGapStart := vPrevEnd;
  vGapEnd   := ioTask[iTrans].Queue[qi].StartTime;

  IF vGapEnd > vGapStart + LINT#1 THEN
    si := si + 1;
    IF si <= DEP_MAX_IDLE_SLOTS THEN
      ioIdleSlot[iTrans].Slots[si].StartTime   := vGapStart;
      ioIdleSlot[iTrans].Slots[si].EndTime     := vGapEnd;
      ioIdleSlot[iTrans].Slots[si].LiftStationTarget := vPrevSink;
      ioIdleSlot[iTrans].Slots[si].SinkStationTarget := ioTask[iTrans].Queue[qi].LiftStationTarget;
    END_IF;
  END_IF;

  vPrevEnd  := ioTask[iTrans].Queue[qi].FinishTime;
  vPrevSink := ioTask[iTrans].Queue[qi].SinkStationTarget;
END_FOR;

si := si + 1;
IF si <= DEP_MAX_IDLE_SLOTS THEN
  ioIdleSlot[iTrans].Slots[si].StartTime   := vPrevEnd;
  ioIdleSlot[iTrans].Slots[si].EndTime     := HORIZON;
  ioIdleSlot[iTrans].Slots[si].LiftStationTarget := vPrevSink;
  ioIdleSlot[iTrans].Slots[si].SinkStationTarget := 0;
END_IF;

ioIdleSlot[iTrans].Count := si;
FC_DEP_CalcIdleSlots := TRUE;

END_FUNCTION

(* ---- FC_DEP_CalcOverlap.st ---- *)
(* ===========================================================================================
 *  FC_DEP_CalcOverlap — Overlap station detection
 *
 *  Company : Galvatek part of the John Cockerill Group
 *  Author  : Jarmo Piipponen
 *  Created : 25.03.2026
 *
 * -------------------------------------------------------------------------------------------
 *  Identifies stations vCovered by 2+ transporters.
 *  Reads Transporters (read-only config). Writes ioOverlap.
 *
 *  ------------------------------------------------------------------------------------------
 *
 *  Changes:
 *
 *
 *
 *)

FUNCTION FC_DEP_CalcOverlap : BOOL

(* Introduction of Variables ----------------------------------------------------------------*)

VAR_IN_OUT
  ioOverlap                : UDT_JC_DepOverlapType;
END_VAR

VAR_EXTERNAL CONSTANT
    MAX_TRANSPORTERS        : INT;
    MIN_STATION_INDEX        : INT;
    MAX_STATION_INDEX        : INT;
END_VAR

VAR_EXTERNAL
  Transporters                     : ARRAY[0..MAX_TRANSPORTERS] OF UDT_TransporterType;
END_VAR

VAR
  vStationIdx               : INT;
  ti                        : INT;
  ai                        : INT;
  vCoverCount               : INT;
  vCovered                   : BOOL;
  vArea                      : UDT_TaskAreaType;
END_VAR

ioOverlap.Count := 0;

FOR vStationIdx := 0 TO 200 DO
  ioOverlap.Flags[vStationIdx] := FALSE;
END_FOR;

FOR vStationIdx := MIN_STATION_INDEX TO MAX_STATION_INDEX DO
  vCoverCount := 0;

  FOR ti := 1 TO MAX_TRANSPORTERS DO
    vCovered := FALSE;
    FOR ai := 1 TO 4 DO
      IF NOT vCovered THEN
        vArea := Transporters[ti].TaskArea[ai];
        IF (vArea.MinLift > 0 AND vStationIdx >= vArea.MinLift AND vStationIdx <= vArea.MaxLift)
           OR (vArea.MinSink > 0 AND vStationIdx >= vArea.MinSink AND vStationIdx <= vArea.MaxSink) THEN
          vCovered := TRUE;
        END_IF;
      END_IF;
    END_FOR;
    IF vCovered THEN
      vCoverCount := vCoverCount + 1;
    END_IF;
  END_FOR;

  IF vCoverCount >= 2 THEN
    ioOverlap.Flags[vStationIdx] := TRUE;
    ioOverlap.Count := ioOverlap.Count + 1;
  END_IF;
END_FOR;

FC_DEP_CalcOverlap := TRUE;

END_FUNCTION

(* ---- FC_DEP_FitTaskToSlot.st ---- *)
(* ===========================================================================================
 *  FC_DEP_FitTaskToSlot — Fit a departure task into idle slots
 *
 *  Company : Galvatek part of the John Cockerill Group
 *  Author  : Jarmo Piipponen
 *  Created : 25.03.2026
 *
 * -------------------------------------------------------------------------------------------
 *  Reads idle slots and move times.
 *  Returns fit result via VAR_OUTPUT.
 *
 *  ------------------------------------------------------------------------------------------
 *
 *  Changes:
 *
 *
 *
 *)

FUNCTION FC_DEP_FitTaskToSlot : BOOL

(* Introduction of Variables ----------------------------------------------------------------*)

VAR_INPUT
  iLiftStn                : INT;
  iSinkStn                : INT;
  iTransId                : INT;
  iTaskStart              : LINT;
  iTaskEnd                : LINT;
  iShiftS                 : REAL;
  iCalcTimeS             : DINT;
  iMinTimeS              : DINT;
  iMaxTimeS              : DINT;
  iFlexFactor             : REAL;
  iMarginS                : REAL;
  iConflictMarginS       : REAL;
END_VAR

VAR_IN_OUT  (* array sizes must match GVL_JC_Constants: 3=MAX_TRANSPORTERS *)
  ioIdleSlot              : ARRAY[1..3] OF UDT_JC_DepIdleSlotSetType;
  ioResult                  : UDT_JC_DepFitResultType;
END_VAR

VAR_EXTERNAL CONSTANT
    MAX_TRANSPORTERS        : INT;
    DEP_MAX_IDLE_SLOTS      : INT;
    SCH_DISPATCH_MARGIN_S   : REAL;
END_VAR

VAR_EXTERNAL
  g_move                    : ARRAY[1..MAX_TRANSPORTERS] OF UDT_JC_MoveTimesType;
END_VAR

VAR
  vSi                        : INT;
  vSlotCnt                  : INT;
  vSlotStart                : LINT;
  vSlotEnd                  : LINT;
  vFromStn                  : INT;
  vToStn                    : INT;
  vTravelTo                 : REAL;
  vTravelFrom               : REAL;
  vEarliest                  : LINT;
  vLatest                    : LINT;
  vTaskDur                  : LINT;
  vDelay                     : REAL;
  vFlexUp                   : REAL;
  vCappedFlex               : REAL;
  vBestDelay                : REAL;
  vBestSlot                 : INT;
  vFound                     : BOOL;
  vOverflowBestDelay       : REAL;
  vOverflowBestSlot        : INT;
  vTmpMove                  : UDT_JC_MoveTimesType;
  vTotalDelay               : REAL;
END_VAR

ioResult.Fits         := FALSE;
ioResult.DelayTime    := 0;
ioResult.NeedExtraTime := 0;
ioResult.TaskEndTime  := 0;
ioResult.SlotIdx      := 0;
ioResult.OverflowSlotIdx := 0;
ioResult.TransporterId := iTransId;
FC_DEP_FitTaskToSlot := FALSE;

IF iTransId < 1 OR iTransId > MAX_TRANSPORTERS THEN RETURN; END_IF;

vTaskDur   := iTaskEnd - iTaskStart;
(* Absolute cap: flex based on full (max - min) range, not (max - calc).
   This prevents cumulative drift when CalcTime is vAdjusted across rounds. *)
vFlexUp    := DINT_TO_REAL(iMaxTimeS - iMinTimeS);
  IF vFlexUp < 0.0 THEN vFlexUp := 0.0; END_IF;
vCappedFlex := vFlexUp * iFlexFactor;

vSlotCnt   := ioIdleSlot[iTransId].Count;
vBestDelay := 1.0E9;
vBestSlot  := 0;
vFound      := FALSE;
vOverflowBestDelay := 1.0E9;
vOverflowBestSlot  := 0;

vTmpMove := g_move[iTransId];
FOR vSi := 1 TO DEP_MAX_IDLE_SLOTS DO
  IF vSi > vSlotCnt THEN EXIT; END_IF;

  vSlotStart := ioIdleSlot[iTransId].Slots[vSi].StartTime;
  vSlotEnd   := ioIdleSlot[iTransId].Slots[vSi].EndTime;

  vFromStn := ioIdleSlot[iTransId].Slots[vSi].LiftStationTarget;
  vTravelTo := 0.0;
  IF vFromStn > 0 AND vFromStn <> iLiftStn THEN
    vTravelTo := FC_STC_CalcHorizontalTravel(iFromStn := vFromStn, iToStn := iLiftStn, iMove := vTmpMove);
  END_IF;

  vToStn := ioIdleSlot[iTransId].Slots[vSi].SinkStationTarget;
  vTravelFrom := 0.0;
  IF vToStn > 0 AND vToStn <> iSinkStn THEN
    vTravelFrom := FC_STC_CalcHorizontalTravel(iFromStn := iSinkStn, iToStn := vToStn, iMove := vTmpMove);
  END_IF;

  (* vEarliest = max(transporter arrival, task readiness) + vConflict margin *)
  IF (vSlotStart + REAL_TO_LINT(vTravelTo)) > (iTaskStart + REAL_TO_LINT(iShiftS)) THEN
    vEarliest := vSlotStart + REAL_TO_LINT(vTravelTo + iConflictMarginS);
  ELSE
    vEarliest := iTaskStart + REAL_TO_LINT(iShiftS + iConflictMarginS);
  END_IF;

  IF vSlotEnd > LINT#9000000000 THEN
    vLatest := LINT#9000000000;
  ELSE
    vLatest := vSlotEnd - REAL_TO_LINT(vTravelFrom + SCH_DISPATCH_MARGIN_S);
  END_IF;

  IF vEarliest + vTaskDur <= vLatest THEN
    vDelay := LINT_TO_REAL(vEarliest - iTaskStart) - iShiftS;
  IF vDelay < 0.0 THEN vDelay := 0.0; END_IF;
    vTotalDelay := iShiftS + vDelay;

    IF vTotalDelay <= iMarginS OR vTotalDelay <= vCappedFlex + 1.0 THEN
      IF vDelay < vBestDelay THEN
        vBestDelay := vDelay;
        vBestSlot  := vSi;
        vFound      := TRUE;
      END_IF;
    ELSE
      IF vDelay < vOverflowBestDelay THEN
        vOverflowBestDelay := vDelay;
        vOverflowBestSlot  := vSi;
      END_IF;
    END_IF;
  END_IF;
END_FOR;

IF vFound THEN
  ioResult.Fits      := TRUE;
  ioResult.DelayTime := REAL_TO_DINT(vBestDelay);
  ioResult.SlotIdx   := vBestSlot;
  ioResult.TaskEndTime := iTaskStart + REAL_TO_LINT(iShiftS + vBestDelay) + vTaskDur;
  ioResult.NeedExtraTime := 0;
ELSE
  ioResult.Fits := FALSE;
  IF vOverflowBestDelay < 1.0E8 THEN
    ioResult.DelayTime     := REAL_TO_DINT(vOverflowBestDelay);
    ioResult.NeedExtraTime := REAL_TO_DINT(iShiftS + vOverflowBestDelay - vCappedFlex);
  IF ioResult.NeedExtraTime < 0 THEN ioResult.NeedExtraTime := 0; END_IF;
    ioResult.OverflowSlotIdx := vOverflowBestSlot;
  ELSE
    ioResult.NeedExtraTime := 0;
  END_IF;
END_IF;

FC_DEP_FitTaskToSlot := TRUE;

END_FUNCTION

(* ---- FC_DEP_OverlapDelay.st ---- *)
(* ===========================================================================================
 *  FC_DEP_OverlapDelay — Overlap vConflict vDelay calculation
 *
 *  Company : Galvatek part of the John Cockerill Group
 *  Author  : Jarmo Piipponen
 *  Created : 25.03.2026
 *
 * -------------------------------------------------------------------------------------------
 *  Returns vDelay vNeeded to avoid overlap conflicts.
 *  Reads task queues via ioTask (sandbox or live).
 *
 *  ------------------------------------------------------------------------------------------
 *
 *  Changes:
 *
 *
 *
 *)

FUNCTION FC_DEP_OverlapDelay : REAL   (* returns delay_s, 0 = no vConflict *)

(* Introduction of Variables ----------------------------------------------------------------*)

VAR_INPUT
  iLiftStn                : INT;
  iSinkStn                : INT;
  iTransId                : INT;
  iTaskStart              : LINT;
  iTaskEnd                : LINT;
  iMarginS                : REAL;
END_VAR

VAR_IN_OUT  (* array sizes must match GVL_JC_Constants: 3=MAX_TRANSPORTERS *)
  ioTask                   : ARRAY[1..3] OF UDT_JC_TskQueueType;
  ioOverlap                : UDT_JC_DepOverlapType;
END_VAR

VAR_EXTERNAL CONSTANT
    MAX_TRANSPORTERS        : INT;
    MAX_UNITS               : INT;
    DEP_MAX_DELAY_ACTS      : INT;
END_VAR

VAR
  vLiftIsOverlap           : BOOL;
  vSinkIsOverlap           : BOOL;
  vRound                     : INT;
  vTi                        : INT;
  vQi                        : INT;
  vMaxConf                  : REAL;
  vTStart                   : LINT;
  vTEnd                     : LINT;
  vEStart                   : LINT;
  vEEnd                     : LINT;
  vELift                    : INT;
  vESink                    : INT;
  vHasOvlp                  : BOOL;
  vNeeded                    : REAL;
  vDelay                     : REAL;
END_VAR

vDelay := 0.0;

IF iLiftStn >= 0 AND iLiftStn <= 200 THEN
  vLiftIsOverlap := ioOverlap.Flags[iLiftStn];
ELSE
  vLiftIsOverlap := FALSE;
END_IF;
IF iSinkStn >= 0 AND iSinkStn <= 200 THEN
  vSinkIsOverlap := ioOverlap.Flags[iSinkStn];
ELSE
  vSinkIsOverlap := FALSE;
END_IF;

IF NOT vLiftIsOverlap AND NOT vSinkIsOverlap THEN
  FC_DEP_OverlapDelay := 0.0;
  RETURN;
END_IF;

FOR vRound := 1 TO DEP_MAX_DELAY_ACTS DO
  vMaxConf := 0.0;
  vTStart  := iTaskStart + REAL_TO_LINT(vDelay);
  vTEnd    := iTaskEnd + REAL_TO_LINT(vDelay);

  FOR vTi := 1 TO MAX_TRANSPORTERS DO
    IF vTi <> iTransId THEN
      FOR vQi := 1 TO MAX_UNITS DO
        IF vQi > ioTask[vTi].Count THEN EXIT; END_IF;

        vELift  := ioTask[vTi].Queue[vQi].LiftStationTarget;
        vESink  := ioTask[vTi].Queue[vQi].SinkStationTarget;
        vEStart := ioTask[vTi].Queue[vQi].StartTime;
        vEEnd   := ioTask[vTi].Queue[vQi].FinishTime;

        vHasOvlp := FALSE;
        IF vELift >= 0 AND vELift <= 200 THEN
  IF ioOverlap.Flags[vELift] THEN vHasOvlp := TRUE; END_IF;
        END_IF;
        IF NOT vHasOvlp AND vESink >= 0 AND vESink <= 200 THEN
  IF ioOverlap.Flags[vESink] THEN vHasOvlp := TRUE; END_IF;
        END_IF;

        IF vHasOvlp THEN
          IF vTStart < (vEEnd + REAL_TO_LINT(iMarginS)) AND vTEnd > (vEStart - REAL_TO_LINT(iMarginS)) THEN
            vNeeded := LINT_TO_REAL(vEEnd - vTStart) + iMarginS;
  IF vNeeded > vMaxConf THEN vMaxConf := vNeeded; END_IF;
          END_IF;
        END_IF;

      END_FOR;
    END_IF;
  END_FOR;

  IF vMaxConf <= 0.0 THEN EXIT; END_IF;
  vDelay := vDelay + vMaxConf;
END_FOR;

FC_DEP_OverlapDelay := vDelay;

END_FUNCTION

(* ---- FC_DEP_Sandbox.st ---- *)
(* ===========================================================================================
 *  FC_DEP_Sandbox — Sandbox snapshot / restore / clear
 *
 *  Company : Galvatek part of the John Cockerill Group
 *  Author  : Jarmo Piipponen
 *  Created : 25.03.2026
 *
 * -------------------------------------------------------------------------------------------
 *  Copies batch and program data between live globals and
 *  DEP workspace arrays via VAR_IN_OUT.
 *  Schedule is NOT copied — DEP calculates it fresh (phases 1000+i).
 *  Task queues are NOT copied — DEP rebuilds them (phases 2000+).
 *
 *  Commands:
 *  1 = SNAPSHOT  — live batch+program → workspace
 *  2 = RESTORE   — workspace batch+program → live
 *  3 = CLEAR     — noop for array-based workspace
 *
 *  ------------------------------------------------------------------------------------------
 *
 *  Changes:
 *
 *
 *
 *)

FUNCTION FC_DEP_Sandbox : BOOL

(* Introduction of Variables ----------------------------------------------------------------*)

VAR_INPUT
  iCmd                     : INT;
END_VAR

VAR_IN_OUT  (* array sizes must match GVL_JC_Constants: 10=MAX_UNITS, 3=MAX_TRANSPORTERS *)
  ioWkSchedule            : ARRAY[1..10] OF UDT_JC_TskScheduleType;
  ioWkBatch               : ARRAY[1..10] OF UDT_BatchType;
  ioWkProgram             : ARRAY[1..10] OF UDT_TreatmentProgramType;
  ioWkTask                : ARRAY[1..3] OF UDT_JC_TskQueueType;
END_VAR

VAR_EXTERNAL CONSTANT
    MAX_TRANSPORTERS        : INT;
    MAX_UNITS               : INT;
END_VAR

VAR_EXTERNAL
  g_schedule                : ARRAY[1..MAX_UNITS] OF UDT_JC_TskScheduleType;
  g_batch                   : ARRAY[1..MAX_UNITS] OF UDT_BatchType;
  TreatmentPrograms                 : ARRAY[1..MAX_UNITS] OF UDT_TreatmentProgramType;
  g_task                    : ARRAY[1..MAX_TRANSPORTERS] OF UDT_JC_TskQueueType;
END_VAR

VAR
  ui                        : INT;
END_VAR

FC_DEP_Sandbox := TRUE;

IF iCmd = 1 THEN
  (* SNAPSHOT: clear workspace, then copy live batch+program *)
  FOR ui := 1 TO MAX_UNITS DO
    ioWkSchedule[ui].StageCount := 0;
    ioWkBatch[ui]    := g_batch[ui];
    ioWkProgram[ui]  := TreatmentPrograms[ui];
  END_FOR;
  FOR ui := 1 TO MAX_TRANSPORTERS DO
    ioWkTask[ui].Count := 0;
  END_FOR;
ELSIF iCmd = 2 THEN
  (* RESTORE: workspace batch+program → live (for REJECT rollback) *)
  FOR ui := 1 TO MAX_UNITS DO
    IF ioWkBatch[ui].BatchCode > 0 THEN
      g_batch[ui] := ioWkBatch[ui];
    END_IF;
    IF ioWkProgram[ui].ProgramId > 0 THEN
      TreatmentPrograms[ui] := ioWkProgram[ui];
    END_IF;
  END_FOR;
ELSIF iCmd = 3 THEN
  ;  (* CLEAR: nothing vNeeded *)

END_IF;

END_FUNCTION

(* ---- FC_STC_CalcHorizontalTravel.st ---- *)
(* ===========================================================================================
 *  FC_STC_CalcHorizontalTravel — Horizontal vTravel time
 *
 *  Company : Galvatek part of the John Cockerill Group
 *  Author  : Jarmo Piipponen
 *  Created : 25.03.2026
 *
 * -------------------------------------------------------------------------------------------
 *  Calculates horizontal vTravel time between two stations
 *  (no lift/sink) using precomputed move time table.
 *  Caller passes iMove (UDT_JC_MoveTimesType) for the
 *  specific transporter.
 *
 *  ------------------------------------------------------------------------------------------
 *
 *  Changes:
 *
 *
 *
 *)

FUNCTION FC_STC_CalcHorizontalTravel : REAL

(* Introduction of Variables ----------------------------------------------------------------*)

VAR_INPUT
  iFromStn                : INT;     (* source station number *)
  iToStn                  : INT;     (* destination station number *)
  iMove                    : UDT_JC_MoveTimesType;   (* transporter's precomputed move times *)
END_VAR

VAR
  vFromIdx                  : INT;
  vToIdx                    : INT;
END_VAR

FC_STC_CalcHorizontalTravel := 0.0;
IF iFromStn > 0 AND iToStn > 0 AND iFromStn <> iToStn THEN
  vFromIdx := iFromStn - MIN_STATION_INDEX;
  vToIdx   := iToStn - MIN_STATION_INDEX;
  IF vFromIdx >= 1 AND vFromIdx <= 25 AND vToIdx >= 1 AND vToIdx <= 25 THEN
    FC_STC_CalcHorizontalTravel := INT_TO_REAL(iMove.Travel[vFromIdx].ToTime[vToIdx]) / 10.0;
  END_IF;
END_IF;

END_FUNCTION

(* ---- FC_STC_CalcSchedule.st ---- *)
(* ===========================================================================================
 *  FC_STC_CalcSchedule — Calculate batch schedule for one unit
 *
 *  Company : Galvatek part of the John Cockerill Group
 *  Author  : Jarmo Piipponen
 *  Created : 25.03.2026
 *
 * -------------------------------------------------------------------------------------------
 *  Shared FC: both TSK and DEP call this with different arrays.
 *  Calculates start/finish times for each treatment stage based
 *  on elapsed time, cal_time and transfer durations.
 *
 *  ------------------------------------------------------------------------------------------
 *
 *  Changes:
 *
 *
 *
 *)

FUNCTION FC_STC_CalcSchedule : BOOL

(* Introduction of Variables ----------------------------------------------------------------*)

VAR_INPUT
  i_unit                    : INT;
  i_trans                   : INT;
  i_time_s                  : LINT;
END_VAR

VAR_IN_OUT  (* array sizes must match GVL_JC_Constants: 10=MAX_UNITS *)
  io_schedule               : ARRAY[1..10] OF UDT_JC_TskScheduleType;
  io_batch                  : ARRAY[1..10] OF UDT_BatchType;
  io_program                : ARRAY[1..10] OF UDT_TreatmentProgramType;
END_VAR

VAR_EXTERNAL CONSTANT
    MIN_STATION_INDEX        : INT;
    MAX_STATION_INDEX        : INT;
    MAX_UNITS               : INT;
    MAX_TRANSPORTERS        : INT;
    MAX_STEPS_PER_PROGRAM   : INT;
    NOT_PROCESSED           : INT;
    USED                    : INT;
END_VAR

VAR_EXTERNAL
  g_unit                    : ARRAY[1..MAX_UNITS] OF UDT_JC_UnitType;
  Stations                 : ARRAY[MIN_STATION_INDEX..MAX_STATION_INDEX] OF UDT_StationType;
  g_station_occupancy             : ARRAY[1..MAX_STATION_INDEX] OF UDT_JC_UnitAtStationType;
  CountStations              : INT;
  g_move                    : ARRAY[1..MAX_TRANSPORTERS] OF UDT_JC_MoveTimesType;
  Transporters                     : ARRAY[0..MAX_TRANSPORTERS] OF UDT_TransporterType;
  g_transporter             : ARRAY[1..MAX_TRANSPORTERS] OF UDT_TransporterStatusType;
END_VAR

VAR
  stg                       : INT;
  stn_num                   : INT;
  prev_stn                  : INT;
  cur_stage                 : INT;
  location                  : INT;
  start_st                  : INT;
  entry_t                   : LINT;
  exit_t                    : LINT;
  xfer_t                    : REAL;
  calc_s                    : REAL;
  min_s                     : REAL;
  max_s                     : REAL;
  is_on_stn                 : BOOL;
  is_first                  : BOOL;
  remain_s                  : REAL;
  elapsed_s                 : REAL;
  p                         : INT;
  chosen_stn                : INT;
  tmp_move                  : UDT_JC_MoveTimesType;
  cand_arr                  : ARRAY[1..5] OF INT;
  cand_cnt                  : INT;
  sched_occupied            : ARRAY[1..5] OF BOOL;
  best_change_time          : LINT;
  my_entry                  : LINT;
  my_exit                   : LINT;
  ov_start                  : LINT;
  ov_end                    : LINT;
  uj                        : INT;
  sj                        : INT;
END_VAR

FC_STC_CalcSchedule := FALSE;
IF i_unit < 1 OR i_unit > MAX_UNITS THEN RETURN; END_IF;
IF i_trans < 1 OR i_trans > MAX_TRANSPORTERS THEN RETURN; END_IF;

cur_stage := io_batch[i_unit].CurStage;
location  := g_unit[i_unit].location;
is_on_stn := location >= MIN_STATION_INDEX;

(* Clear old schedule *)
FOR stg := 0 TO MAX_STEPS_PER_PROGRAM DO
  io_schedule[i_unit].Stages[stg].Station := 0;
  io_schedule[i_unit].Stages[stg].ProgramStage := 0;
  io_schedule[i_unit].Stages[stg].EntryTime := 0;
  io_schedule[i_unit].Stages[stg].ExitTime := 0;
  io_schedule[i_unit].Stages[stg].MinTime := 0;
  io_schedule[i_unit].Stages[stg].CalcTime := 0;
  io_schedule[i_unit].Stages[stg].MaxTime := 0;
  io_schedule[i_unit].Stages[stg].TransferTime := 0;
END_FOR;
io_schedule[i_unit].StageCount := 0;

(* Waiting batch (state = NOT_PROCESSED): treat as stage 0 *)
IF io_batch[i_unit].State = NOT_PROCESSED THEN
  cur_stage := 0;
END_IF;

IF is_on_stn THEN
  start_st := cur_stage;
ELSE
  start_st := cur_stage + 1;
END_IF;
IF start_st < 1 THEN
  start_st := 1;
END_IF;

IF is_on_stn THEN
  prev_stn := location;
ELSIF cur_stage >= 1 AND cur_stage <= 30 THEN
  prev_stn := io_program[i_unit].Steps[cur_stage].Stations[0];
ELSE
  prev_stn := 0;
END_IF;

exit_t := i_time_s;
is_first := TRUE;

(* Prepend current location to Stages[0] when unit needs pre-positioning *)
IF is_on_stn AND start_st >= 1 THEN
  stn_num := 0;
  FOR p := 0 TO 4 DO
    IF io_program[i_unit].Steps[start_st].Stations[p] = location THEN
      stn_num := location;
    END_IF;
  END_FOR;
  IF stn_num = 0 THEN
    io_schedule[i_unit].Stages[0].Station       := location;
    io_schedule[i_unit].Stages[0].ProgramStage := 0;
    io_schedule[i_unit].Stages[0].EntryTime    := exit_t;
    io_schedule[i_unit].Stages[0].TransferTime := 0;

    IF io_batch[i_unit].CurStage = 0 AND io_batch[i_unit].CalTime > 0 THEN
      IF io_batch[i_unit].StartTime > 0 AND io_batch[i_unit].StartTime < i_time_s THEN
        elapsed_s := LINT_TO_REAL(i_time_s - io_batch[i_unit].StartTime);
      ELSE
        elapsed_s := 0.0;
      END_IF;
      remain_s := DINT_TO_REAL(io_batch[i_unit].CalTime) - elapsed_s;
  IF remain_s < 1.0 THEN remain_s := 1.0; END_IF;
      exit_t := i_time_s + REAL_TO_LINT(remain_s);
      io_schedule[i_unit].Stages[0].ExitTime  := exit_t;
      io_schedule[i_unit].Stages[0].CalcTime  := REAL_TO_DINT(remain_s);
      io_schedule[i_unit].Stages[0].MinTime   := io_batch[i_unit].MinTime;
      io_schedule[i_unit].Stages[0].MaxTime   := io_batch[i_unit].MaxTime;
    ELSE
      (* Pickup wait: transporter horizontal travel time to this station, min 5s *)
      calc_s := FC_STC_CalcHorizontalTravel(
        i_from_stn := g_transporter[i_trans].CurrentStation,
        i_to_stn   := location,
        i_move     := g_move[i_trans]);
      IF calc_s < 5.0 THEN calc_s := 5.0; END_IF;
      exit_t := i_time_s + REAL_TO_LINT(calc_s);
      io_schedule[i_unit].Stages[0].ExitTime  := exit_t;
      io_schedule[i_unit].Stages[0].CalcTime  := REAL_TO_DINT(calc_s);
      io_schedule[i_unit].Stages[0].MinTime   := REAL_TO_DINT(calc_s);
      io_schedule[i_unit].Stages[0].MaxTime   := REAL_TO_DINT(2.0 * calc_s);
    END_IF;

    is_first := FALSE;
  END_IF;
END_IF;

(* ============================================================
   MAIN LOOP: Calculate schedule for each program stage
   ============================================================ *)
FOR stg := start_st TO io_program[i_unit].StepCount DO

  cand_cnt := 0;
  FOR p := 0 TO 4 DO
    IF io_program[i_unit].Steps[stg].Stations[p] > 0 THEN
      cand_cnt := cand_cnt + 1;
      cand_arr[cand_cnt] := io_program[i_unit].Steps[stg].Stations[p];
      sched_occupied[cand_cnt] := FALSE;
    END_IF;
  END_FOR;

  IF cand_cnt = 0 THEN
    EXIT;
  END_IF;

  chosen_stn := 0;
  IF is_first AND is_on_stn AND stg = cur_stage THEN
    FOR p := 1 TO cand_cnt DO
      IF cand_arr[p] = location THEN
        chosen_stn := location;
      END_IF;
    END_FOR;
  END_IF;

  IF chosen_stn = 0 THEN
    IF cand_cnt = 1 THEN
      chosen_stn := cand_arr[1];
    ELSE
      (* Estimate this batch's time window per candidate for overlap check *)
      calc_s := DINT_TO_REAL(io_program[i_unit].Steps[stg].CalTime);
      tmp_move := g_move[i_trans];

      FOR p := 1 TO cand_cnt DO
        (* Calculate entry/exit per candidate station individually *)
        xfer_t := FC_STC_CalcTransferTime(
          i_from_stn            := prev_stn,
          i_to_stn              := cand_arr[p],
          i_move                := tmp_move,
          i_from_dropping_x10   := Stations[prev_stn].DrippingTime,
          i_to_device_delay_x10 := Stations[cand_arr[p]].DeviceDelay,
          i_drip_tray_delay_x10 := Transporters[i_trans].DripTrayDelay
        );
        my_entry := exit_t + REAL_TO_LINT(xfer_t);
        my_exit  := my_entry + REAL_TO_LINT(calc_s);

        FOR uj := 1 TO MAX_UNITS DO
          IF uj <> i_unit AND io_schedule[uj].StageCount > 0 THEN
            FOR sj := 0 TO io_schedule[uj].StageCount DO
              IF io_schedule[uj].Stages[sj].Station = cand_arr[p] THEN
                ov_start := my_entry;
                IF io_schedule[uj].Stages[sj].EntryTime > ov_start THEN
                  ov_start := io_schedule[uj].Stages[sj].EntryTime;
                END_IF;
                ov_end := my_exit;
                IF io_schedule[uj].Stages[sj].ExitTime < ov_end THEN
                  ov_end := io_schedule[uj].Stages[sj].ExitTime;
                END_IF;
                IF ov_end > ov_start THEN
                  sched_occupied[p] := TRUE;
                END_IF;
              END_IF;
            END_FOR;
          END_IF;
        END_FOR;

      END_FOR;

      (* Pass 1: prefer schedule-free station, pick earliest ChangeTime *)
      best_change_time := LINT#9999999999;
      FOR p := 1 TO cand_cnt DO
        IF NOT sched_occupied[p] THEN
          IF cand_arr[p] >= MIN_STATION_INDEX AND cand_arr[p] <= MAX_STATION_INDEX THEN
            IF g_station_occupancy[cand_arr[p]].ChangeTime < best_change_time THEN
              best_change_time := g_station_occupancy[cand_arr[p]].ChangeTime;
              chosen_stn := cand_arr[p];
            END_IF;
          END_IF;
        END_IF;
      END_FOR;

      (* Pass 2: all sched-occupied — pick first candidate *)
      IF chosen_stn = 0 THEN
        chosen_stn := cand_arr[1];
      END_IF;
    END_IF;
  END_IF;

  stn_num := chosen_stn;

  calc_s := DINT_TO_REAL(io_program[i_unit].Steps[stg].CalTime);
  min_s  := DINT_TO_REAL(io_program[i_unit].Steps[stg].MinTime);
  max_s  := DINT_TO_REAL(io_program[i_unit].Steps[stg].MaxTime);

  tmp_move := g_move[i_trans];
  IF prev_stn >= MIN_STATION_INDEX AND prev_stn <= MAX_STATION_INDEX
     AND stn_num >= MIN_STATION_INDEX AND stn_num <= MAX_STATION_INDEX THEN
    IF Stations[prev_stn].Crosstransport > 0
       AND Stations[prev_stn].ChangeStation > 0
       AND Stations[prev_stn].YPosition <> Stations[stn_num].YPosition THEN
      xfer_t := INT_TO_REAL(Stations[prev_stn].CrossTransportTime)
              + FC_STC_CalcTransferTime(
                  i_from_stn            := Stations[prev_stn].ChangeStation,
                  i_to_stn              := stn_num,
                  i_move                := tmp_move,
                  i_from_dropping_x10   := Stations[Stations[prev_stn].ChangeStation].DrippingTime,
                  i_to_device_delay_x10 := Stations[stn_num].DeviceDelay,
                  i_drip_tray_delay_x10 := Transporters[i_trans].DripTrayDelay
                );
    ELSE
      xfer_t := FC_STC_CalcTransferTime(
        i_from_stn            := prev_stn,
        i_to_stn              := stn_num,
        i_move                := tmp_move,
        i_from_dropping_x10   := Stations[prev_stn].DrippingTime,
        i_to_device_delay_x10 := Stations[stn_num].DeviceDelay,
        i_drip_tray_delay_x10 := Transporters[i_trans].DripTrayDelay
      );
    END_IF;
  ELSE
    xfer_t := 60.0;
  END_IF;

  IF is_first AND is_on_stn AND stg = cur_stage THEN
    entry_t := i_time_s;
    IF io_batch[i_unit].StartTime > 0 THEN
      elapsed_s := LINT_TO_REAL(i_time_s - io_batch[i_unit].StartTime);
    ELSE
      elapsed_s := 0.0;
    END_IF;
    remain_s := DINT_TO_REAL(io_batch[i_unit].CalTime) - elapsed_s;
  IF remain_s < 1.0 THEN remain_s := 1.0; END_IF;
    exit_t := i_time_s + REAL_TO_LINT(remain_s);
  ELSIF is_first AND NOT is_on_stn THEN
    IF io_batch[i_unit].StartTime > 0 AND io_batch[i_unit].CalTime > 0 THEN
      entry_t := io_batch[i_unit].StartTime + DINT_TO_LINT(io_batch[i_unit].CalTime);
    ELSE
      entry_t := i_time_s + REAL_TO_LINT(xfer_t);
    END_IF;
    exit_t  := entry_t + REAL_TO_LINT(calc_s);
  ELSE
    entry_t := exit_t + REAL_TO_LINT(xfer_t);
    exit_t  := entry_t + REAL_TO_LINT(calc_s);
  END_IF;

  IF stg <= 30 THEN
    io_schedule[i_unit].Stages[stg].Station       := stn_num;
    io_schedule[i_unit].Stages[stg].ProgramStage := stg;
    io_schedule[i_unit].Stages[stg].EntryTime    := entry_t;
    io_schedule[i_unit].Stages[stg].ExitTime     := exit_t;
    io_schedule[i_unit].Stages[stg].MinTime      := REAL_TO_DINT(min_s);
    io_schedule[i_unit].Stages[stg].CalcTime     := REAL_TO_DINT(calc_s);
    io_schedule[i_unit].Stages[stg].MaxTime      := REAL_TO_DINT(max_s);
    io_schedule[i_unit].Stages[stg].TransferTime := REAL_TO_DINT(xfer_t);
    io_schedule[i_unit].StageCount := stg;
  END_IF;

  prev_stn := stn_num;
  is_first := FALSE;

END_FOR;

FC_STC_CalcSchedule := TRUE;

END_FUNCTION

(* ---- FC_STC_CalcTransferTime.st ---- *)
(* ===========================================================================================
 *  FC_STC_CalcTransferTime — Total transfer time calculation
 *
 *  Company : Galvatek part of the John Cockerill Group
 *  Author  : Jarmo Piipponen
 *  Created : 25.03.2026
 *
 * -------------------------------------------------------------------------------------------
 *  Calculates total transfer time between two stations using
 *  precomputed move time table plus operational delays:
 *  p2 = lift_s  + fromDroppingTime + dripTrayDelay
 *  p3 = travel_s
 *  p4 = sink_s  + dripTrayDelay    + toDeviceDelay
 *
 *  Lift station device_delay is NOT added because covers
 *  are opened during treatment time (overlaps).
 *
 *  All delay inputs are INT ×10 (tenths of second).
 *
 *  ------------------------------------------------------------------------------------------
 *
 *  Changes:
 *
 *
 *
 *)

FUNCTION FC_STC_CalcTransferTime : REAL

(* Introduction of Variables ----------------------------------------------------------------*)

VAR_INPUT
  i_from_stn                : INT;     (* source station, e.g. 105 *)
  i_to_stn                  : INT;     (* destination station, e.g. 112 *)
  i_move                    : UDT_JC_MoveTimesType;   (* transporter's precomputed move times *)
  i_from_dropping_x10       : INT;     (* Stations[from].DrippingTime — tenths of second *)
  i_to_device_delay_x10     : INT;     (* Stations[to].DeviceDelay   — tenths of second *)
  i_drip_tray_delay_x10     : INT;     (* Transporters[trans].DripTrayDelay  — tenths of second *)
END_VAR

VAR
  from_idx                  : INT;
  to_idx                    : INT;
END_VAR

FC_STC_CalcTransferTime := 0.0;
IF i_from_stn > 0 AND i_from_stn <> i_to_stn THEN
  from_idx := i_from_stn - MIN_STATION_INDEX;
  to_idx   := i_to_stn - MIN_STATION_INDEX;
  IF from_idx >= 1 AND from_idx <= 25 AND to_idx >= 1 AND to_idx <= 25 THEN
    FC_STC_CalcTransferTime :=
      (* Phase 2: lift + dropping + drip tray *)
      INT_TO_REAL(i_move.LiftTime[from_idx]) / 10.0
      + INT_TO_REAL(i_from_dropping_x10) / 10.0
      + INT_TO_REAL(i_drip_tray_delay_x10) / 10.0
      (* Phase 3: horizontal travel *)
      + INT_TO_REAL(i_move.Travel[from_idx].ToTime[to_idx]) / 10.0
      (* Phase 4: sink + drip tray + device delay *)
      + INT_TO_REAL(i_move.SinkTime[to_idx]) / 10.0
      + INT_TO_REAL(i_drip_tray_delay_x10) / 10.0
      + INT_TO_REAL(i_to_device_delay_x10) / 10.0;
  END_IF;
END_IF;

END_FUNCTION

(* ---- FC_STC_CollectActiveBatches.st ---- *)
(* ===========================================================================================
 *  FC_STC_CollectActiveBatches — Filter active/waiting batches
 *
 *  Company : Galvatek part of the John Cockerill Group
 *  Author  : Jarmo Piipponen
 *  Created : 25.03.2026
 *
 * -------------------------------------------------------------------------------------------
 *  Returns count of matching batches; fills oList via VAR_OUTPUT.
 *
 *  Mode:
 *  iMode = 0 — active (in-production) batches
 *  iMode = 1 — waiting batches (station 114 lookup)
 *
 *  ------------------------------------------------------------------------------------------
 *
 *  Changes:
 *
 *
 *
 *)

FUNCTION FC_STC_CollectActiveBatches : INT   (* returns count *)

(* Introduction of Variables ----------------------------------------------------------------*)

VAR_INPUT
  iMode : INT;    (* 0 = all active, 1 = waiting only *)
END_VAR

VAR_EXTERNAL CONSTANT
    MAX_UNITS         : INT;
    MAX_STATION_INDEX : INT;
    USED              : INT;
    TO_NONE           : INT;
    NOT_PROCESSED     : INT;
    IN_PROCESS        : INT;
END_VAR

VAR_EXTERNAL
  gBatch            : ARRAY[1..MAX_UNITS] OF UDT_BatchType;
  gUnit             : ARRAY[1..MAX_UNITS] OF UDT_JC_UnitType;
  TreatmentPrograms : ARRAY[1..MAX_UNITS] OF UDT_TreatmentProgramType;
  gStationOccupancy : ARRAY[1..MAX_STATION_INDEX] OF UDT_JC_UnitAtStationType;
END_VAR

VAR_OUTPUT
  oList : ARRAY[1..MAX_UNITS] OF INT;  (* unit indices *)
END_VAR

VAR
  vUi  : INT;
  vCnt : INT;
END_VAR

vCnt := 0;
FOR vUi := 1 TO MAX_UNITS DO
  oList[vUi] := 0;
END_FOR;

IF iMode = 1 THEN
  (* ── Waiting batch: direct lookup at station 114 ── *)
  vUi := gStationOccupancy[114].UnitId;
  IF vUi >= 1 AND vUi <= MAX_UNITS THEN
    IF gUnit[vUi].Status = USED
       AND gUnit[vUi].Target = TO_NONE
       AND gBatch[vUi].State = NOT_PROCESSED
       AND gBatch[vUi].ProgId = TreatmentPrograms[vUi].ProgramId
       AND TreatmentPrograms[vUi].ProgramId > 0 THEN
      vCnt := 1;
      oList[1] := vUi;
    END_IF;
  END_IF;
  FC_STC_CollectActiveBatches := vCnt;
  RETURN;
END_IF;

(* ── Mode 0: active batches — loop ── *)
FOR vUi := 1 TO MAX_UNITS DO
  IF gUnit[vUi].Status = USED
     AND gUnit[vUi].Target = TO_NONE
     AND gBatch[vUi].ProgId = TreatmentPrograms[vUi].ProgramId
     AND TreatmentPrograms[vUi].ProgramId > 0 THEN

    IF gBatch[vUi].State = IN_PROCESS
       AND gBatch[vUi].CurStage >= 0
       AND gBatch[vUi].CurStage <= 99 THEN
      vCnt := vCnt + 1;
      oList[vCnt] := vUi;
    END_IF;
  END_IF;
END_FOR;

FC_STC_CollectActiveBatches := vCnt;

END_FUNCTION

(* ---- FC_STC_CreateTasks.st ---- *)
(* ===========================================================================================
 *  FC_STC_CreateTasks — Build task list from schedule for one unit
 *
 *  Company : Galvatek part of the John Cockerill Group
 *  Author  : Jarmo Piipponen
 *  Created : 25.03.2026
 *
 * -------------------------------------------------------------------------------------------
 *  Shared FC: both TSK and DEP call this with different arrays.
 *  Creates transporter tasks from the calculated schedule stages
 *  and appends them to the task queues.
 *
 *  ------------------------------------------------------------------------------------------
 *
 *  Changes:
 *
 *
 *
 *)

FUNCTION FC_STC_CreateTasks : BOOL

(* Introduction of Variables ----------------------------------------------------------------*)

VAR_INPUT
  i_unit                    : INT;
END_VAR

VAR_IN_OUT  (* array sizes must match GVL_JC_Constants: 10=MAX_UNITS, 3=MAX_TRANSPORTERS *)
  io_schedule               : ARRAY[1..10] OF UDT_JC_TskScheduleType;
  io_task                   : ARRAY[1..3] OF UDT_JC_TskQueueType;
END_VAR

VAR_EXTERNAL CONSTANT
    MAX_TRANSPORTERS        : INT;
    MAX_UNITS               : INT;
    MAX_TASK_QUEUE          : INT;
    MIN_STATION_INDEX        : INT;
    MAX_STATION_INDEX        : INT;
END_VAR

VAR_EXTERNAL
  Transporters                     : ARRAY[0..MAX_TRANSPORTERS] OF UDT_TransporterType;
  Stations                 : ARRAY[MIN_STATION_INDEX..MAX_STATION_INDEX] OF UDT_StationType;
END_VAR

VAR
  si                        : INT;
  sc                        : INT;
  lift_stn                  : INT;
  sink_stn                  : INT;
  tid                       : INT;
  qi                        : INT;
  fb_find                   : FB_STC_FindTransporter;
  eff_lift_stn              : INT;
END_VAR

FC_STC_CreateTasks := FALSE;
IF i_unit < 1 OR i_unit > MAX_UNITS THEN RETURN; END_IF;

sc := io_schedule[i_unit].StageCount;
IF sc < 1 THEN RETURN; END_IF;

(* Start from 0 if Stages[0] exists (prepend), else from 1 *)
FOR si := 0 TO sc - 1 DO
  IF io_schedule[i_unit].Stages[si].Station = 0 THEN
    (* Skip unused stage slot *)
  ELSE
    lift_stn := io_schedule[i_unit].Stages[si].Station;
    sink_stn := io_schedule[i_unit].Stages[si + 1].Station;

    IF lift_stn > 0 AND sink_stn > 0 THEN
      eff_lift_stn := lift_stn;
      IF lift_stn >= MIN_STATION_INDEX AND lift_stn <= MAX_STATION_INDEX
         AND sink_stn >= MIN_STATION_INDEX AND sink_stn <= MAX_STATION_INDEX THEN
        IF Stations[lift_stn].Crosstransport > 0
           AND Stations[lift_stn].ChangeStation > 0
           AND Stations[lift_stn].YPosition <> Stations[sink_stn].YPosition THEN
          eff_lift_stn := Stations[lift_stn].ChangeStation;
        END_IF;
      END_IF;

      fb_find(i_lift_stn := eff_lift_stn, i_sink_stn := sink_stn);
      tid := fb_find.o_trans;

      IF tid >= 1 AND tid <= 3 THEN
        qi := io_task[tid].Count + 1;
        IF qi <= MAX_TASK_QUEUE THEN
          io_task[tid].Queue[qi].Unit         := i_unit;
          io_task[tid].Queue[qi].Stage        := io_schedule[i_unit].Stages[si + 1].ProgramStage;
          io_task[tid].Queue[qi].SrcStage     := io_schedule[i_unit].Stages[si].ProgramStage;
          io_task[tid].Queue[qi].LiftStationTarget := eff_lift_stn;
          io_task[tid].Queue[qi].SinkStationTarget := sink_stn;
          io_task[tid].Queue[qi].StartTime   := io_schedule[i_unit].Stages[si].ExitTime;
          io_task[tid].Queue[qi].FinishTime  := io_schedule[i_unit].Stages[si + 1].EntryTime;
          io_task[tid].Queue[qi].CalcTime    := io_schedule[i_unit].Stages[si].CalcTime;
          io_task[tid].Queue[qi].MinTime     := io_schedule[i_unit].Stages[si].MinTime;
          io_task[tid].Queue[qi].MaxTime     := io_schedule[i_unit].Stages[si].MaxTime;
          io_task[tid].Count := qi;
        END_IF;
      END_IF;
    END_IF;
  END_IF; (* skip unused stage slot *)
END_FOR;

FC_STC_CreateTasks := TRUE;

END_FUNCTION

(* ---- FC_STC_DispatchTask.st ---- *)
(* ===========================================================================================
 *  FC_STC_DispatchTask — Validate and dispatch tasks to transporters
 *
 *  Company : Galvatek part of the John Cockerill Group
 *  Author  : Jarmo Piipponen
 *  Created : 25.03.2026
 *
 * -------------------------------------------------------------------------------------------
 *  Called every PLC scan from MainScheduler.
 *  For each idle transporter with queued tasks:
 *  1. Skip if transporter not idle or queue empty
 *  2. Time check: start_time close enough?
 *  3. Sink station free check (with parallel alternatives)
 *  4. Conflict check against active transporters
 *  5. Dispatch: write to g_transporter → RunTasks picks it up
 *
 *  ------------------------------------------------------------------------------------------
 *
 *  Changes:
 *
 *
 *
 *)

FUNCTION FC_STC_DispatchTask : BOOL

(* Introduction of Variables ----------------------------------------------------------------*)

VAR_EXTERNAL CONSTANT
    MAX_TRANSPORTERS        : INT;
    MAX_UNITS               : INT;
    MAX_STATIONS_PER_STEP   : INT;
    MAX_STEPS_PER_PROGRAM   : INT;
    MIN_STATION_INDEX        : INT;
    MAX_STATION_INDEX        : INT;
    SCH_DISPATCH_MARGIN_S   : REAL;
    USED                    : INT;
    PROCESSED               : INT;
END_VAR

VAR_EXTERNAL
  g_transporter             : ARRAY[1..MAX_TRANSPORTERS] OF UDT_TransporterStatusType;
  g_task                    : ARRAY[1..MAX_TRANSPORTERS] OF UDT_JC_TskQueueType;
  Stations                 : ARRAY[MIN_STATION_INDEX..MAX_STATION_INDEX] OF UDT_StationType;
  g_station_occupancy             : ARRAY[1..MAX_STATION_INDEX] OF UDT_JC_UnitAtStationType;
  g_unit                    : ARRAY[1..MAX_UNITS] OF UDT_JC_UnitType;
  TreatmentPrograms                 : ARRAY[1..MAX_UNITS] OF UDT_TreatmentProgramType;
  g_ntt                     : ARRAY[1..MAX_TRANSPORTERS] OF UDT_JC_NttTransporterType;
  g_batch                   : ARRAY[1..MAX_UNITS] OF UDT_BatchType;
  g_move                    : ARRAY[1..MAX_TRANSPORTERS] OF UDT_JC_MoveTimesType;
  Transporters                     : ARRAY[0..MAX_TRANSPORTERS] OF UDT_TransporterType;
  g_schedule                : ARRAY[1..MAX_UNITS] OF UDT_JC_TskScheduleType;
  g_time_s                  : LINT;
  g_event_pending           : UDT_JC_EventMsgType;
  g_event_pending_valid     : BOOL;
  g_dispatched_task         : ARRAY[1..MAX_TRANSPORTERS] OF UDT_JC_DispatchedTaskType;
END_VAR

VAR
  ti                        : INT;     (* transporter loop *)
  (* Task fields — read from queue[1] to avoid struct copy *)
  t_unit                    : INT;
  t_stage                   : INT;
  t_lift                    : INT;
  t_sink                    : INT;
  t_start                   : LINT;
  t_finish                  : LINT;
  t_calc_time               : DINT;
  (* Time check *)
  travel_s                  : REAL;
  margin_s                  : LINT;
  from_idx                  : INT;
  to_idx                    : INT;
  (* Sink search *)
  sink_stn                  : INT;
  sink_free                 : BOOL;
  best_stn                  : INT;
  best_change               : LINT;
  si                        : INT;
  cand_stn                  : INT;
  cand_free                 : BOOL;
  uj                        : INT;
  tgt                       : INT;
  ntt_idx                   : INT;     (* resolved NTT index (buffer 6/7/8) *)
  ntt_cnt                   : INT;
  ntt_fb_cnt                : INT;
  (* Conflict check *)
  conflict                  : BOOL;
  cj                        : INT;
  task_min                  : INT;     (* min station of our proposed task *)
  task_max                  : INT;     (* max station of our proposed task *)
  (* Queue position loop *)
  qi                        : INT;
  (* Shift-down after dispatch *)
  sh                        : INT;
  (* Transfer time for batch progress bar *)
  xfer_total                : REAL;
  (* Program stage number for event *)
  prog_stage                : INT;
  (* Manual task dispatch flag *)
  unit_ok                   : BOOL;
END_VAR

FOR ti := 1 TO MAX_TRANSPORTERS DO

  (* ── 1. Skip if not idle or queue empty ── *)
  (* Accept idle (Phase=0) OR move-away in progress (Phase=1, Status=3) *)
  IF (g_transporter[ti].Phase = 0 OR (g_transporter[ti].Phase = 1 AND g_transporter[ti].Status = 3))
     AND g_task[ti].Count >= 1 THEN

    (* Try each queue position — skip blocked tasks, dispatch first feasible *)
    FOR qi := 1 TO g_task[ti].Count DO

    (* Read task fields from queue position qi *)
    t_unit      := g_task[ti].Queue[qi].Unit;
    t_stage     := g_task[ti].Queue[qi].Stage;  (* schedule index *)
    t_lift      := g_task[ti].Queue[qi].LiftStationTarget;
    t_sink      := g_task[ti].Queue[qi].SinkStationTarget;
    t_start     := g_task[ti].Queue[qi].StartTime;
    t_finish    := g_task[ti].Queue[qi].FinishTime;
    t_calc_time := g_task[ti].Queue[qi].CalcTime;

    (* Queue[].Stage already contains ProgramStage (set by FC_STC_CreateTasks) *)
    prog_stage := t_stage;

    (* ── 1b. Lift station unit check — unit must be AT the lift station ── *)
    (* Manual tasks have Unit=0 → skip unit-location check *)
    (* NOTE: CODESYS does NOT short-circuit OR — use nested IFs *)
    unit_ok := FALSE;
    IF t_unit = 0 THEN
      unit_ok := TRUE;
    ELSIF t_unit >= 1 AND t_unit <= MAX_UNITS THEN
      IF g_unit[t_unit].location = t_lift THEN
        unit_ok := TRUE;
      END_IF;
    END_IF;

    IF unit_ok THEN

    (* ── 2. Time check ── *)
    travel_s := 0.0;
    IF g_transporter[ti].CurrentStation > 0 AND t_lift > 0
       AND g_transporter[ti].CurrentStation <> t_lift THEN
      from_idx := g_transporter[ti].CurrentStation - MIN_STATION_INDEX;
      to_idx   := t_lift - MIN_STATION_INDEX;
      IF from_idx >= 1 AND from_idx <= 30 AND to_idx >= 1 AND to_idx <= 30 THEN
        travel_s := INT_TO_REAL(g_move[ti].Travel[from_idx].ToTime[to_idx]) / 10.0;
      END_IF;
    END_IF;

    margin_s := t_start - g_time_s;

    IF margin_s <= REAL_TO_LINT(travel_s + SCH_DISPATCH_MARGIN_S) THEN

      (* ── 3. Sink station free check ── *)
      sink_stn := t_sink;
      sink_free := FALSE;

      IF sink_stn >= MIN_STATION_INDEX AND sink_stn <= MAX_STATION_INDEX THEN
        sink_free := TRUE;
        FOR uj := 1 TO MAX_UNITS DO
          IF g_unit[uj].location = sink_stn AND g_unit[uj].Status = USED THEN
            sink_free := FALSE;
          END_IF;
        END_FOR;
      END_IF;

      IF NOT sink_free THEN
        (* Search alternative parallel stations *)
        best_stn := 0;
        best_change := LINT#2000000000;

        IF prog_stage >= 1 AND prog_stage <= MAX_STEPS_PER_PROGRAM
           AND t_unit >= 1 AND t_unit <= MAX_UNITS THEN
          (* Treatment task — look in TreatmentPrograms for parallel stations *)
          FOR si := 0 TO MAX_STATIONS_PER_STEP - 1 DO
            cand_stn := TreatmentPrograms[t_unit].Steps[prog_stage].Stations[si];
            IF cand_stn > 0 AND cand_stn <> t_sink THEN
              IF cand_stn >= MIN_STATION_INDEX AND cand_stn <= MAX_STATION_INDEX THEN
                cand_free := TRUE;
                FOR uj := 1 TO MAX_UNITS DO
                  IF g_unit[uj].location = cand_stn AND g_unit[uj].Status = USED THEN
                    cand_free := FALSE;
                  END_IF;
                END_FOR;
                IF cand_free THEN
                  IF g_station_occupancy[cand_stn].ChangeTime < best_change THEN
                    best_change := g_station_occupancy[cand_stn].ChangeTime;
                    best_stn := cand_stn;
                  END_IF;
                END_IF;
              END_IF;
            END_IF;
          END_FOR;

        ELSIF prog_stage = 0 AND t_unit >= 1 AND t_unit <= MAX_UNITS THEN
          (* No-treatment task — look in g_ntt for alternatives *)
          tgt := g_unit[t_unit].Target;
          IF tgt >= 1 AND tgt <= 5 THEN
            (* Resolve buffer NTT index like NoTreatment does *)
            IF tgt = 2 THEN
              IF g_batch[t_unit].BatchCode = 0 THEN
                ntt_idx := 6;
              ELSIF g_batch[t_unit].State = PROCESSED THEN
                ntt_idx := 8;
              ELSE
                ntt_idx := 7;
              END_IF;
            ELSE
              ntt_idx := tgt;
            END_IF;
            (* Check primary stations *)
            ntt_cnt := g_ntt[ti].Target[ntt_idx].StationCount;
            FOR si := 1 TO ntt_cnt DO
              IF si <= MAX_STATIONS_PER_STEP THEN
                cand_stn := g_ntt[ti].Target[ntt_idx].Stations[si];
                IF cand_stn > 0 AND cand_stn <> t_sink THEN
                  IF cand_stn >= MIN_STATION_INDEX AND cand_stn <= MAX_STATION_INDEX THEN
                    cand_free := TRUE;
                    FOR uj := 1 TO MAX_UNITS DO
                      IF g_unit[uj].location = cand_stn AND g_unit[uj].Status = USED THEN
                        cand_free := FALSE;
                      END_IF;
                    END_FOR;
                    IF cand_free THEN
                      IF g_station_occupancy[cand_stn].ChangeTime < best_change THEN
                        best_change := g_station_occupancy[cand_stn].ChangeTime;
                        best_stn := cand_stn;
                      END_IF;
                    END_IF;
                  END_IF;
                END_IF;
              END_IF;
            END_FOR;
            (* Check fallback stations *)
            ntt_fb_cnt := g_ntt[ti].Target[ntt_idx].FallbackCount;
            FOR si := 1 TO ntt_fb_cnt DO
              IF si <= MAX_STATIONS_PER_STEP THEN
                cand_stn := g_ntt[ti].Target[ntt_idx].FallbackStations[si];
                IF cand_stn > 0 AND cand_stn <> t_sink THEN
                  IF cand_stn >= MIN_STATION_INDEX AND cand_stn <= MAX_STATION_INDEX THEN
                    cand_free := TRUE;
                    FOR uj := 1 TO MAX_UNITS DO
                      IF g_unit[uj].location = cand_stn AND g_unit[uj].Status = USED THEN
                        cand_free := FALSE;
                      END_IF;
                    END_FOR;
                    IF cand_free THEN
                      IF g_station_occupancy[cand_stn].ChangeTime < best_change THEN
                        best_change := g_station_occupancy[cand_stn].ChangeTime;
                        best_stn := cand_stn;
                      END_IF;
                    END_IF;
                  END_IF;
                END_IF;
              END_IF;
            END_FOR;
          END_IF;
        END_IF;

        IF best_stn > 0 THEN
          sink_stn := best_stn;
          sink_free := TRUE;
        END_IF;
      END_IF;  (* NOT sink_free *)

      IF sink_free THEN

        (* ── 4. Conflict check ── *)
        conflict := FALSE;

        IF t_lift <= sink_stn THEN
          task_min := t_lift;
          task_max := sink_stn;
        ELSE
          task_min := sink_stn;
          task_max := t_lift;
        END_IF;

        FOR cj := 1 TO MAX_TRANSPORTERS DO
          IF cj <> ti AND g_transporter[cj].Phase > 0 THEN

            (* a) T2's entire active task inside our range → conflict *)
            IF g_transporter[cj].LiftStationTarget >= task_min
               AND g_transporter[cj].LiftStationTarget <= task_max
               AND g_transporter[cj].SinkStationTarget >= task_min
               AND g_transporter[cj].SinkStationTarget <= task_max THEN
              conflict := TRUE;
            END_IF;

            (* b) T2 delivers to one of our exact stations → conflict *)
            IF g_transporter[cj].SinkStationTarget = t_lift
               OR g_transporter[cj].SinkStationTarget = sink_stn THEN
              conflict := TRUE;
            END_IF;

          END_IF;
        END_FOR;

        IF NOT conflict THEN
          (* ── 5. Dispatch: assign task to transporter ── *)
          g_transporter[ti].TaskId      := t_start;
          g_transporter[ti].LiftStationTarget := t_lift;
          g_transporter[ti].SinkStationTarget := sink_stn;
          g_transporter[ti].CurrentTaskFinishTime := g_task[ti].Queue[qi].FinishTime;
          g_station_occupancy[ti].UnitId      := t_unit;
          g_transporter[ti].TaskRemainingTime := t_calc_time;

          (* ── 5b. Fill dispatched task package ── *)
          g_dispatched_task[ti].TaskId           := t_start;
          g_dispatched_task[ti].UnitId           := t_unit;
          g_dispatched_task[ti].LiftStation      := t_lift;
          g_dispatched_task[ti].SinkStation      := sink_stn;
          IF t_lift >= MIN_STATION_INDEX AND t_lift <= MAX_STATION_INDEX THEN
            g_dispatched_task[ti].LiftX              := Stations[t_lift].XPosition;
            g_dispatched_task[ti].LiftKind           := Stations[t_lift].DryWet;
            g_dispatched_task[ti].DroppingTime_x10   := Stations[t_lift].DrippingTime;
            g_dispatched_task[ti].LiftDeviceDelay_x10 := Stations[t_lift].DeviceDelay;
          END_IF;
          IF sink_stn >= MIN_STATION_INDEX AND sink_stn <= MAX_STATION_INDEX THEN
            g_dispatched_task[ti].SinkX              := Stations[sink_stn].XPosition;
            g_dispatched_task[ti].SinkKind           := Stations[sink_stn].DryWet;
            g_dispatched_task[ti].SinkDeviceDelay_x10 := Stations[sink_stn].DeviceDelay;
          END_IF;
          g_dispatched_task[ti].DripTrayDelay_x10 := Transporters[ti].DripTrayDelay;
          g_dispatched_task[ti].TreatmentTime    := t_calc_time;
          g_dispatched_task[ti].MinTime          := g_task[ti].Queue[qi].MinTime;
          g_dispatched_task[ti].MaxTime          := g_task[ti].Queue[qi].MaxTime;
          g_dispatched_task[ti].NttPrimary       := g_task[ti].Queue[qi].NttPrimary;
          IF t_unit >= 1 AND t_unit <= MAX_UNITS THEN
            g_dispatched_task[ti].BatchCode      := g_batch[t_unit].BatchCode;
            g_dispatched_task[ti].ProgramStage   := g_batch[t_unit].CurStage;
          ELSE
            g_dispatched_task[ti].BatchCode      := 0;
            g_dispatched_task[ti].ProgramStage   := 0;
          END_IF;
          g_dispatched_task[ti].Active           := TRUE;

          (* ── Emit TASK_DISPATCHED event (msg_type=1) ── *)
          xfer_total := FC_STC_CalcTransferTime(
            i_from_stn            := t_lift,
            i_to_stn              := sink_stn,
            i_move                := g_move[ti],
            i_from_dropping_x10   := Stations[t_lift].DrippingTime,
            i_to_device_delay_x10 := Stations[sink_stn].DeviceDelay,
            i_drip_tray_delay_x10 := Transporters[ti].DripTrayDelay
          );
          IF xfer_total < 1.0 THEN
            xfer_total := INT_TO_REAL(ABS(sink_stn - t_lift)) * 8.0;
          END_IF;
  IF xfer_total < 5.0 THEN xfer_total := 60.0; END_IF;
          g_dispatched_task[ti].TransferTime_x10 := REAL_TO_DINT(xfer_total * 10.0);
          IF NOT g_event_pending_valid THEN
            g_event_pending.MsgType := 1;
            g_event_pending.TsHi := LINT_TO_UINT(g_time_s / LINT#65536);
            g_event_pending.TsLo := LINT_TO_UINT(g_time_s MOD LINT#65536);
            g_event_pending.Payload[1]  := LINT_TO_INT(t_start / LINT#65536);   (* TaskId_Hi *)
            g_event_pending.Payload[2]  := LINT_TO_INT(t_start MOD LINT#65536);  (* TaskId_Lo *)
            g_event_pending.Payload[3]  := ti;
            g_event_pending.Payload[4]  := t_unit;
            g_event_pending.Payload[5]  := t_lift;
            g_event_pending.Payload[6]  := sink_stn;
            IF t_unit >= 1 AND t_unit <= MAX_UNITS THEN
              prog_stage := g_batch[t_unit].CurStage;
              g_event_pending.Payload[7]  := prog_stage;
              g_event_pending.Payload[8]  := g_batch[t_unit].BatchCode;
            ELSE
              g_event_pending.Payload[7]  := 0;
              g_event_pending.Payload[8]  := 0;
            END_IF;
            g_event_pending.Payload[9]  := DINT_TO_INT(t_calc_time);
            g_event_pending.Payload[10] := DINT_TO_INT(g_task[ti].Queue[qi].MinTime);
            g_event_pending.Payload[11] := DINT_TO_INT(g_task[ti].Queue[qi].MaxTime);
            g_event_pending.Payload[12] := REAL_TO_INT(xfer_total);
            g_event_pending_valid := TRUE;
          END_IF;

          (* Copy station-specific timing from config *)
          IF t_lift >= MIN_STATION_INDEX AND t_lift <= MAX_STATION_INDEX THEN
            g_transporter[ti].DrippingTime := Stations[t_lift].DrippingTime;
          END_IF;

          (* Shift queue: remove position qi, move rest up *)
          FOR sh := qi + 1 TO g_task[ti].Count DO
            g_task[ti].Queue[sh - 1] := g_task[ti].Queue[sh];
          END_FOR;
          (* Clear last slot *)
          g_task[ti].Queue[g_task[ti].Count].Unit := 0;
          g_task[ti].Queue[g_task[ti].Count].Stage := 0;
          g_task[ti].Queue[g_task[ti].Count].SrcStage := 0;
          g_task[ti].Queue[g_task[ti].Count].LiftStationTarget := 0;
          g_task[ti].Queue[g_task[ti].Count].SinkStationTarget := 0;
          g_task[ti].Queue[g_task[ti].Count].StartTime := 0;
          g_task[ti].Queue[g_task[ti].Count].FinishTime := 0;
          g_task[ti].Queue[g_task[ti].Count].CalcTime := 0;
          g_task[ti].Queue[g_task[ti].Count].MinTime := 0;
          g_task[ti].Queue[g_task[ti].Count].MaxTime := 0;
          g_task[ti].Count := g_task[ti].Count - 1;
          EXIT;  (* dispatched — stop searching this queue *)

        END_IF;  (* NOT conflict *)

      END_IF;  (* sink_free *)

    END_IF;  (* time check *)

    END_IF;  (* unit at lift station *)

    END_FOR;  (* qi — try next queue position *)

  END_IF;  (* idle + queue *)

END_FOR;

FC_STC_DispatchTask := TRUE;

END_FUNCTION
